// ---------- recipe writes (READY only, bounds-checked) ----------
parToggle := GVL_Cmd.mbParRegs[3];
IF (parToggle <> lastParTog) AND (GVL_Sts.mode = E_MachMode.READY) THEN
    lastParTog := parToggle;
    itemP := WORD_TO_INT(GVL_Cmd.mbParRegs[0]);
    cookP := TO_LREAL(WORD_TO_INT(GVL_Cmd.mbParRegs[1])) / 10.0;
    setP  := TO_LREAL(WORD_TO_INT(GVL_Cmd.mbParRegs[2])) / 10.0;
    IF (itemP >= 1) AND (itemP <= 4)
       AND (cookP >= 20.0) AND (cookP <= 300.0)
       AND (setP >= 120.0) AND (setP <= 230.0) THEN
        GVL_Par.aRecipe[itemP].cookTimeS  := cookP;
        GVL_Par.aRecipe[itemP].platenSetC := setP;
    END_IF
END_IF

END_PROGRAM

// Device/Application/05_L4_Comms/PRG_HMI
(* ============================================================
   PRG_HMI — HMI request edges + password-gated jog (T_Comms).
   Buttons arrive as GVL_Cmd.hmi* (mapped to HMI tags at site).
   NOTE: in the SFC/LD refactor this POU's edge networks become
   LD rungs one-per-button (technician-facing).
   ============================================================ *)
PROGRAM PRG_HMI
VAR
    rtStart, rtStop, rtReset, rtAck, rtClean : R_TRIG;
    jogPermit : BOOL;
    jogStep   : LREAL;
    tonJog    : TON;
    MAINT_PIN : UINT := 2468;   // TODO site-specific, move to secure store
    rtRecW, rtTrimW : R_TRIG;
    recOk   : BOOL;
    recIt   : INT;
    recV    : LREAL;
    trimP   : INT;
    bJogP, bJogM : BOOL;         // jog levels (direct var OR HMI register bit)
    wFlags  : WORD;
    it2, z2, base : INT;
    rtPrsW  : R_TRIG;            // press service command
    prsSel  : INT;
    prsHold : INT;               // holds CmdExec for a few comms cycles
    prsView : INT;               // press shown on the status page
END_VAR

// ---------- LT2100E register unpack (HMI writes %MW600..609) ----------
// reg[0] button bits: 0=start 1=stop 2=reset 3=ack 4=clean
//                     5=jog+ 6=jog- 7=recipeWrite 8=trimWrite
// Numerics are copied only while their write/jog bit is held, so direct
// variable writes (watch list / sim testing) keep working unchanged.
IF GVL_Cmd.hmiRegsCmd[1] <> 0 THEN
    GVL_Cmd.hmiMaintPin := TO_UINT(GVL_Cmd.hmiRegsCmd[1]);
END_IF
IF (GVL_Cmd.hmiRegsCmd[0] AND 16#0060) <> 0 THEN            // a jog bit is held
    GVL_Cmd.hmiJogAxis := TO_INT(GVL_Cmd.hmiRegsCmd[2]);
END_IF
IF (GVL_Cmd.hmiRegsCmd[0] AND 16#0080) <> 0 THEN            // recipe write
    GVL_Cmd.hmiRecItem  := TO_UINT(GVL_Cmd.hmiRegsCmd[3]);
    GVL_Cmd.hmiRecField := TO_UINT(GVL_Cmd.hmiRegsCmd[4]);
    GVL_Cmd.hmiRecValue := TO_LREAL(GVL_Cmd.hmiRegsCmd[5]) / 10.0;   // x10 scaling
END_IF
IF (GVL_Cmd.hmiRegsCmd[0] AND 16#0100) <> 0 THEN            // trim write
    GVL_Cmd.hmiTrimPress := TO_UINT(GVL_Cmd.hmiRegsCmd[6]);
    GVL_Cmd.hmiTrimDelta := TO_LREAL(TO_INT(GVL_Cmd.hmiRegsCmd[7])) / 100.0;  // x100 signed
END_IF
bJogP := GVL_Cmd.hmiJogPlus  OR ((GVL_Cmd.hmiRegsCmd[0] AND 16#0020) <> 0);
bJogM := GVL_Cmd.hmiJogMinus OR ((GVL_Cmd.hmiRegsCmd[0] AND 16#0040) <> 0);

rtStart(CLK := GVL_Cmd.hmiStart OR ((GVL_Cmd.hmiRegsCmd[0] AND 16#0001) <> 0));
rtStop (CLK := GVL_Cmd.hmiStop  OR ((GVL_Cmd.hmiRegsCmd[0] AND 16#0002) <> 0));
rtReset(CLK := GVL_Cmd.hmiReset OR ((GVL_Cmd.hmiRegsCmd[0] AND 16#0004) <> 0));
rtAck  (CLK := GVL_Cmd.hmiAck   OR ((GVL_Cmd.hmiRegsCmd[0] AND 16#0008) <> 0));
rtClean(CLK := GVL_Cmd.hmiClean OR ((GVL_Cmd.hmiRegsCmd[0] AND 16#0010) <> 0));

GVL_Cmd.reqStart  := rtStart.Q;
GVL_Cmd.reqStop   := rtStop.Q  OR GVL_Cmd.reqStop;    // JobExec may also set; consumed by Supervisor edge
GVL_Cmd.reqReset  := rtReset.Q;
GVL_Cmd.reqAckAll := rtAck.Q;
GVL_Cmd.reqClean  := rtClean.Q OR GVL_Cmd.reqClean;
// self-clearing one-shot semantics: Supervisor uses R_TRIG on these,
// so clear them after one comms cycle
IF NOT rtStop.Q  THEN GVL_Cmd.reqStop  := FALSE; END_IF
IF NOT rtClean.Q THEN GVL_Cmd.reqClean := FALSE; END_IF

// ---------- jog (maintenance only) ----------
jogPermit := (GVL_Cmd.hmiMaintPin = MAINT_PIN)
         AND ((GVL_Sts.mode = E_MachMode.READY) OR (GVL_Sts.mode = E_MachMode.FAULT))
         AND GVL_Sts.safetyOk;
tonJog(IN := jogPermit AND (bJogP OR bJogM), PT := T#100MS);
IF tonJog.Q THEN
    tonJog(IN := FALSE);
    jogStep := LIMIT(1.0, GVL_Par.jogVel, GVL_Cfg.JOG_VEL_MAX) * 0.1;  // mm per 100 ms
    IF bJogM THEN jogStep := -jogStep; END_IF
    CASE GVL_Cmd.hmiJogAxis OF
        1: IF NOT GVL_Mech.axGX.Busy THEN
               GVL_Mech.axGX.TargetPos := GVL_Mech.axGX.Sts.actPos + jogStep;
               GVL_Mech.axGX.Vel := GVL_Par.jogVel;
               GVL_Mech.axGX.MoveExec := TRUE;
           END_IF
        2: IF NOT GVL_Mech.axGT.Busy THEN
               GVL_Mech.axGT.TargetPos := GVL_Mech.axGT.Sts.actPos + jogStep;
               GVL_Mech.axGT.Vel := GVL_Par.jogVel;
               GVL_Mech.axGT.MoveExec := TRUE;
           END_IF
        3: IF NOT GVL_Mech.axGZ.Busy THEN
               GVL_Mech.axGZ.TargetPos := GVL_Mech.axGZ.Sts.actPos + jogStep;
               GVL_Mech.axGZ.Vel := GVL_Par.jogVel;
               GVL_Mech.axGZ.MoveExec := TRUE;
           END_IF
        // axes 4..8: same pattern for scraper X/Y/Z, fork Z/tele — add as needed
    END_CASE
ELSIF NOT (bJogP OR bJogM) THEN
    GVL_Mech.axGX.MoveExec := FALSE;
    GVL_Mech.axGT.MoveExec := FALSE;
    GVL_Mech.axGZ.MoveExec := FALSE;
END_IF

// ---------- press jog (jog axis select 9 = selected press drive) ----------
// Level-driven; the drive FB only jogs while fully idle. Velocity = Pr6.00.
IF (GVL_Cmd.hmiJogAxis = 9) AND jogPermit THEN
    GVL_Mech.drvPress[TO_INT(LIMIT(0, GVL_Cmd.hmiPressSel, 3))].JogPlus  := bJogP;
    GVL_Mech.drvPress[TO_INT(LIMIT(0, GVL_Cmd.hmiPressSel, 3))].JogMinus := bJogM;
ELSE
    FOR it2 := 0 TO 3 DO
        GVL_Mech.drvPress[it2].JogPlus  := FALSE;
        GVL_Mech.drvPress[it2].JogMinus := FALSE;
    END_FOR
END_IF

// ---------- recipe editor (bounds-checked; rejected while RUN) ----------
rtRecW(CLK := GVL_Cmd.hmiRecWrite OR ((GVL_Cmd.hmiRegsCmd[0] AND 16#0080) <> 0));
IF rtRecW.Q THEN
    GVL_Cmd.hmiRecAck := FALSE; GVL_Cmd.hmiRecErr := FALSE;
    recIt := TO_INT(GVL_Cmd.hmiRecItem);
    recV  := GVL_Cmd.hmiRecValue;
    recOk := (recIt >= 1) AND (recIt <= 4) AND (GVL_Sts.mode <> E_MachMode.RUN);
    IF recOk THEN
        CASE GVL_Cmd.hmiRecField OF
            1: IF (recV >= GVL_Cfg.REC_COOK_MIN)  AND (recV <= GVL_Cfg.REC_COOK_MAX)
               THEN GVL_Par.aRecipe[recIt].cookTimeS := recV;  ELSE recOk := FALSE; END_IF
            2: IF (recV >= GVL_Cfg.REC_SMDUR_MIN) AND (recV <= GVL_Cfg.REC_SMDUR_MAX)
               THEN GVL_Par.aRecipe[recIt].smashDurS := recV;  ELSE recOk := FALSE; END_IF
            3: IF (recV >= GVL_Cfg.REC_SMPOS_MIN) AND (recV <= GVL_Cfg.REC_SMPOS_MAX)
               THEN GVL_Par.aRecipe[recIt].smashPosMm := recV; ELSE recOk := FALSE; END_IF
            4: IF (recV >= GVL_Cfg.REC_HLPOS_MIN) AND (recV <= GVL_Cfg.REC_HLPOS_MAX)
               THEN GVL_Par.aRecipe[recIt].holdPosMm := recV;  ELSE recOk := FALSE; END_IF
            5: IF (recV >= GVL_Cfg.REC_PLSET_MIN) AND (recV <= GVL_Cfg.REC_PLSET_MAX)
               THEN GVL_Par.aRecipe[recIt].platenSetC := recV; ELSE recOk := FALSE; END_IF
        ELSE
            recOk := FALSE;
        END_CASE
        // physical sanity: hold gap must not be tighter than smash gap
        IF recOk AND (GVL_Par.aRecipe[recIt].holdPosMm < GVL_Par.aRecipe[recIt].smashPosMm) THEN
            GVL_Par.aRecipe[recIt].holdPosMm := GVL_Par.aRecipe[recIt].smashPosMm;
        END_IF
    END_IF
    GVL_Cmd.hmiRecAck := recOk;
    GVL_Cmd.hmiRecErr := NOT recOk;
END_IF

// ---------- press calibration trim (maintenance PIN; not while RUN) ----------
rtTrimW(CLK := GVL_Cmd.hmiTrimWrite OR ((GVL_Cmd.hmiRegsCmd[0] AND 16#0100) <> 0));
IF rtTrimW.Q THEN
    GVL_Cmd.hmiTrimAck := FALSE; GVL_Cmd.hmiTrimErr := FALSE;
    trimP := TO_INT(GVL_Cmd.hmiTrimPress);
    IF (trimP >= 0) AND (trimP <= 3)
       AND (GVL_Cmd.hmiMaintPin = MAINT_PIN)
       AND (GVL_Sts.mode <> E_MachMode.RUN)
       AND (ABS(GVL_Cmd.hmiTrimDelta) <= GVL_Cfg.PRESS_TRIM_MAX_MM) THEN
        GVL_Par.pressTrimMm[trimP] := LIMIT(-GVL_Cfg.PRESS_TRIM_MAX_MM,
            GVL_Par.pressTrimMm[trimP] + GVL_Cmd.hmiTrimDelta,
            GVL_Cfg.PRESS_TRIM_MAX_MM);
        GVL_Cmd.hmiTrimAck := TRUE;
    ELSE
        GVL_Cmd.hmiTrimErr := TRUE;
    END_IF
END_IF

// ---------- press service commands (PIN; READY only; press must be idle) ----------
// HMI: reg608 = command (1 HOME, 2 OPEN, 3 PROFILE), reg609 = press 0..3,
// button bit 9 executes. Do not use while the test suite or Gateway runs.
rtPrsW(CLK := GVL_Cmd.hmiPressWrite OR ((GVL_Cmd.hmiRegsCmd[0] AND 16#0200) <> 0));
IF rtPrsW.Q THEN
    GVL_Cmd.hmiPressAck := FALSE; GVL_Cmd.hmiPressErr := FALSE;
    IF (GVL_Cmd.hmiRegsCmd[0] AND 16#0200) <> 0 THEN
        GVL_Cmd.hmiPressCmd := TO_UINT(GVL_Cmd.hmiRegsCmd[8]);
        GVL_Cmd.hmiPressSel := TO_UINT(GVL_Cmd.hmiRegsCmd[9]);
    END_IF
    prsSel := TO_INT(GVL_Cmd.hmiPressSel);
    IF (prsSel >= 0) AND (prsSel <= 3)
       AND (GVL_Cmd.hmiMaintPin = MAINT_PIN)
       AND (GVL_Sts.mode = E_MachMode.READY)
       AND (NOT GVL_Mech.fbPress[prsSel].Busy)
       AND (NOT GVL_Cmd.testStart) THEN
        CASE GVL_Cmd.hmiPressCmd OF
            1: GVL_Mech.fbPress[prsSel].Cmd.code := GVL_Cfg.MCMD_HOME;
               GVL_Cmd.hmiPressAck := TRUE;
            2: GVL_Mech.fbPress[prsSel].Cmd.code := GVL_Cfg.MCMD_OPEN;
               GVL_Cmd.hmiPressAck := TRUE;
            3: IF GVL_Mech.fbPress[prsSel].IsOpen THEN   // profile only from open
                   GVL_Mech.fbPress[prsSel].Recipe :=
                       GVL_Par.aRecipe[LIMIT(1, TO_INT(GVL_Cmd.hmiRecItem), 4)];
                   GVL_Mech.fbPress[prsSel].Cmd.code := GVL_Cfg.MCMD_PROFILE;
                   GVL_Cmd.hmiPressAck := TRUE;
               ELSE
                   GVL_Cmd.hmiPressErr := TRUE;          // open (cmd 2) first
               END_IF
        ELSE
            GVL_Cmd.hmiPressErr := TRUE;
        END_CASE
        IF GVL_Cmd.hmiPressAck THEN
            GVL_Mech.fbPress[prsSel].CmdExec := TRUE;
            prsHold := 3;                    // release after ~3 comms cycles
        END_IF
    ELSE
        GVL_Cmd.hmiPressErr := TRUE;
    END_IF
END_IF
IF prsHold > 0 THEN
    prsHold := prsHold - 1;
    IF prsHold = 0 THEN
        GVL_Mech.fbPress[TO_INT(LIMIT(0, GVL_Cmd.hmiPressSel, 3))].CmdExec := FALSE;
    END_IF
END_IF

// ---------- LT2100E status pack (HMI reads %MW620..669) ----------
GVL_Cmd.hmiRegsSts[0] := TO_WORD(TO_UINT(GVL_Sts.mode));
wFlags := 0;
IF GVL_Cmd.hmiRecAck    THEN wFlags := wFlags OR 16#0001; END_IF
IF GVL_Cmd.hmiRecErr    THEN wFlags := wFlags OR 16#0002; END_IF
IF GVL_Cmd.hmiTrimAck   THEN wFlags := wFlags OR 16#0004; END_IF
IF GVL_Cmd.hmiTrimErr   THEN wFlags := wFlags OR 16#0008; END_IF
IF GVL_Sts.heatAtSet    THEN wFlags := wFlags OR 16#0010; END_IF
IF GVL_Sts.fridgeAtSet  THEN wFlags := wFlags OR 16#0020; END_IF
IF GVL_Sts.allHomed     THEN wFlags := wFlags OR 16#0040; END_IF
IF GVL_Sts.safetyOk     THEN wFlags := wFlags OR 16#0080; END_IF
IF GVL_Sts.cleanCoolOk  THEN wFlags := wFlags OR 16#0100; END_IF
IF GVL_Cmd.hmiPressAck  THEN wFlags := wFlags OR 16#0200; END_IF
IF GVL_Cmd.hmiPressErr  THEN wFlags := wFlags OR 16#0400; END_IF
GVL_Cmd.hmiRegsSts[1] := wFlags;
GVL_Cmd.hmiRegsSts[2] := TO_WORD(TO_UINT(GVL_Alm.nActive));
GVL_Cmd.hmiRegsSts[3] := TO_WORD(GVL_Alm.aActive[0].id AND 16#FFFF);          // code
GVL_Cmd.hmiRegsSts[4] := TO_WORD(SHR(GVL_Alm.aActive[0].id, 16) AND 16#FFFF); // subsystem
GVL_Cmd.hmiRegsSts[5] := TO_WORD(TO_UINT(GVL_Sts.uptimeS MOD 65536));
// griddle states 626..629
FOR z2 := 0 TO 3 DO
    GVL_Cmd.hmiRegsSts[6 + z2] := TO_WORD(GVL_Sts.aGriddle[z2].state);
END_FOR
// recipe readback 630..649: per item 1..4 -> cook, smashDur, smashPos, holdPos, platenSet (all x10)
FOR it2 := 1 TO 4 DO
    base := 10 + (it2 - 1) * 5;
    GVL_Cmd.hmiRegsSts[base]     := TO_WORD(TO_UINT(GVL_Par.aRecipe[it2].cookTimeS  * 10.0));
    GVL_Cmd.hmiRegsSts[base + 1] := TO_WORD(TO_UINT(GVL_Par.aRecipe[it2].smashDurS  * 10.0));
    GVL_Cmd.hmiRegsSts[base + 2] := TO_WORD(TO_UINT(GVL_Par.aRecipe[it2].smashPosMm * 10.0));
    GVL_Cmd.hmiRegsSts[base + 3] := TO_WORD(TO_UINT(GVL_Par.aRecipe[it2].holdPosMm  * 10.0));
    GVL_Cmd.hmiRegsSts[base + 4] := TO_WORD(TO_UINT(GVL_Par.aRecipe[it2].platenSetC * 10.0));
END_FOR
// press trims 650..653 (x100 signed)
FOR z2 := 0 TO 3 DO
    GVL_Cmd.hmiRegsSts[30 + z2] := TO_WORD(TO_INT(GVL_Par.pressTrimMm[z2] * 100.0));
END_FOR
// temperatures 654..661 platens, 662 fridge (x10)
FOR z2 := 0 TO 7 DO
    GVL_Cmd.hmiRegsSts[34 + z2] := TO_WORD(TO_INT(GVL_Sts.aHeat[z2].actC * 10.0));
END_FOR
GVL_Cmd.hmiRegsSts[42] := TO_WORD(TO_INT(GVL_Sts.fridgeActC * 10.0));
// press service status page 663..667 (selected press)
prsView := TO_INT(LIMIT(0, GVL_Cmd.hmiPressSel, 3));
GVL_Cmd.hmiRegsSts[43] := TO_WORD(GVL_Mech.fbPress[prsView].State);
wFlags := 0;
IF GVL_Mech.drvPress[prsView].Homed    THEN wFlags := wFlags OR 16#0001; END_IF
IF GVL_Mech.fbPress[prsView].IsOpen    THEN wFlags := wFlags OR 16#0002; END_IF
IF GVL_Mech.fbPress[prsView].Holding   THEN wFlags := wFlags OR 16#0004; END_IF
IF GVL_Mech.fbPress[prsView].Busy      THEN wFlags := wFlags OR 16#0008; END_IF
IF GVL_Mech.fbPress[prsView].Error     THEN wFlags := wFlags OR 16#0010; END_IF
IF GVL_Mech.drvPress[prsView].HomeBusy THEN wFlags := wFlags OR 16#0020; END_IF
IF GVL_Mech.drvPress[prsView].ParamsValid THEN wFlags := wFlags OR 16#0040; END_IF
IF GVL_Mech.drvPress[prsView].Busy     THEN wFlags := wFlags OR 16#0080; END_IF
GVL_Cmd.hmiRegsSts[44] := wFlags;
GVL_Cmd.hmiRegsSts[45] := GVL_IO.iMbPrStatus;   // bench drive raw status word
GVL_Cmd.hmiRegsSts[46] := TO_WORD(GVL_Mech.fbPress[prsView].ErrorID AND 16#FFFF);
GVL_Cmd.hmiRegsSts[47] := TO_WORD(SHR(GVL_Mech.fbPress[prsView].ErrorID, 16) AND 16#FFFF);
// jog feedback 668: selected axis actual position, mm/deg x10 (signed)
CASE GVL_Cmd.hmiJogAxis OF
    1: GVL_Cmd.hmiRegsSts[48] := TO_WORD(TO_INT(GVL_Mech.axGX.Sts.actPos * 10.0));
    2: GVL_Cmd.hmiRegsSts[48] := TO_WORD(TO_INT(GVL_Mech.axGT.Sts.actPos * 10.0));
    3: GVL_Cmd.hmiRegsSts[48] := TO_WORD(TO_INT(GVL_Mech.axGZ.Sts.actPos * 10.0));
ELSE
    GVL_Cmd.hmiRegsSts[48] := 0;
END_CASE

END_PROGRAM

// Device/Application/02_L1_Drivers/FB_AxisCtrl
(* ============================================================
   FB_AxisCtrl — single-axis wrapper. The ONLY POU calling MC_*.
   Runs in T_Motion. One instance per axis, body called EVERY cycle.
   SIM: internal kinematic model (trapezoid-less: const-vel ramp).
   REAL: SoftMotion CiA-402 via SM3_Basic.
   ============================================================ *)
FUNCTION_BLOCK FB_AxisCtrl
VAR_INPUT
    Sim       : BOOL;
    SubsysId  : UINT;
    Enable    : BOOL;
    HomeExec  : BOOL;          // level; internally edge-latched
    MoveExec  : BOOL;
    TargetPos : LREAL;
    Vel       : LREAL := 100.0;
    Acc       : LREAL := 500.0;
    StopExec  : BOOL;
    ResetExec : BOOL;
    Abort     : BOOL;
    CycleMs   : LREAL := 4.0;
    SimHomeS  : LREAL := 1.0;  // sim homing duration
END_VAR
VAR_IN_OUT
    Axis : AXIS_REF_SM3;
END_VAR
VAR_OUTPUT
    Sts     : ST_AxisSts;
    Busy    : BOOL;
    Done    : BOOL;            // latched until next exec
    Error   : BOOL;
    ErrorID : UDINT;
END_VAR
VAR
    state     : INT;           // 0 idle 1 homing 2 moving 3 stopping
    rtHome, rtMove, rtReset : R_TRIG;
    tonTO     : TON;
    // sim model
    simPos    : LREAL;
    simTgt    : LREAL;
    simHomeT  : LREAL;
    // real motion FBs
    mcPower   : MC_Power;
    mcHome    : MC_Home;
    mcMove    : MC_MoveAbsolute;
    mcStop    : MC_Stop;
    mcReset   : MC_Reset;
    dtS       : LREAL;
    stepMax   : LREAL;
END_VAR


dtS := CycleMs / 1000.0;
rtHome(CLK := HomeExec);
rtMove(CLK := MoveExec);
rtReset(CLK := ResetExec);

IF Abort THEN
    state := 0; Busy := FALSE;
    tonTO(IN := FALSE);
END_IF

IF rtReset.Q THEN
    Error := FALSE; ErrorID := 0;
END_IF

IF Sim THEN
    // ---------------- SIMULATION MODEL ----------------
    Sts.powered := Enable;
    CASE state OF
        0: // idle
            IF Enable AND rtHome.Q THEN
                state := 1; simHomeT := 0.0; Busy := TRUE; Done := FALSE;
            ELSIF Enable AND Sts.homed AND rtMove.Q THEN
                simTgt := TargetPos; state := 2; Busy := TRUE; Done := FALSE;
                tonTO(IN := FALSE);
            ELSIF Enable AND (NOT Sts.homed) AND rtMove.Q THEN
                Error := TRUE; ErrorID := F_Err(SubsysId, GVL_Cfg.ERR_NOT_HOMED);
            END_IF
        1: // homing
            simHomeT := simHomeT + dtS;
            IF simHomeT >= SimHomeS THEN
                simPos := 0.0; Sts.homed := TRUE;
                state := 0; Busy := FALSE; Done := TRUE;
            END_IF
        2: // moving: constant-velocity approach
            stepMax := Vel * dtS;
            IF ABS(simTgt - simPos) <= stepMax THEN
                simPos := simTgt;
                state := 0; Busy := FALSE; Done := TRUE;
            ELSIF simTgt > simPos THEN
                simPos := simPos + stepMax;
            ELSE
                simPos := simPos - stepMax;
            END_IF
            tonTO(IN := TRUE, PT := GVL_Cfg.TO_AXIS_MOVE);
            IF tonTO.Q THEN
                state := 0; Busy := FALSE; Error := TRUE;
                ErrorID := F_Err(SubsysId, GVL_Cfg.ERR_TIMEOUT);
            END_IF
    END_CASE
    IF StopExec THEN state := 0; Busy := FALSE; END_IF
    Sts.actPos := simPos;
    Sts.inPos  := (state = 0);
ELSE
    // ---------------- REAL HARDWARE (SoftMotion) ----------------
    mcPower(Axis := Axis, Enable := Enable, bRegulatorOn := Enable, bDriveStart := Enable);
    Sts.powered := mcPower.Status;

    mcHome(Axis := Axis, Execute := (rtHome.Q OR mcHome.Busy) AND NOT Abort, Position := 0.0);
    IF mcHome.Done THEN Sts.homed := TRUE; END_IF

    mcMove(Axis := Axis,
           Execute      := (rtMove.Q OR mcMove.Busy) AND NOT Abort AND NOT StopExec,
           Position     := TargetPos,
           Velocity     := Vel,
           Acceleration := Acc,
           Deceleration := Acc);

    mcStop(Axis := Axis, Execute := StopExec OR Abort, Deceleration := Acc * 2.0);
    mcReset(Axis := Axis, Execute := rtReset.Q);

    Busy := mcHome.Busy OR mcMove.Busy;
    IF mcHome.Done OR mcMove.Done THEN Done := TRUE; END_IF
    IF rtHome.Q OR rtMove.Q THEN Done := FALSE; END_IF

    IF mcMove.Error OR mcHome.Error OR mcPower.Error THEN
        Error := TRUE;
        ErrorID := F_Err(SubsysId, GVL_Cfg.ERR_DRIVE);
        Sts.homed := FALSE;              // demand re-home after drive fault
    END_IF
    Sts.actPos := Axis.fSetPosition;     // TODO: use MC_ReadActualPosition if preferred
    Sts.inPos  := NOT Busy;
END_IF

IF NOT Sts.powered THEN Sts.homed := FALSE; END_IF   // power loss clears homed
Sts.errorId := ErrorID;

END_FUNCTION_BLOCK

// Device/Application/02_L1_Drivers/FB_PidHeater
(* ============================================================
   FB_PidHeater — PI + time-proportioned SSR + TC plausibility.
   Call every T_App cycle; internal divider executes PI at 100 ms.
   SIM: first-order plant  dT = (gain*out - (T-Tamb)/tau) * dt
   Independent hardwired thermostat is the REAL protection; the
   over-temp check here is early warning (INFO/ZONE only).
   ============================================================ *)
FUNCTION_BLOCK FB_PidHeater
VAR_INPUT
    Sim          : BOOL;
    ZoneId       : INT;          // 0..7
    Enable       : BOOL;
    SetC         : LREAL := 200.0;
    iTempRaw     : INT;          // 0.1 degC from TC module
    StaggerToken : BOOL;         // may ramp (from FB_HeatBank)
    CycleMs      : LREAL := 20.0;
END_VAR
VAR_OUTPUT
    qSsr    : BOOL;
    Zone    : ST_HeatZone;
    Error   : BOOL;
    ErrorID : UDINT;
END_VAR
VAR
    divCnt   : INT;
    actC     : LREAL;
    lastC    : LREAL;
    err      : LREAL;
    integ    : LREAL;
    outPct   : LREAL;
    pwmT     : LREAL;
    simC     : LREAL := 25.0;
    dtPi     : LREAL := 0.1;
    tcFaultCnt : INT;
    SIM_GAIN : LREAL := 3.5;     // degC/s at 100 %
    SIM_TAU  : LREAL := 60.0;
    ramping  : BOOL;
END_VAR

// ---- acquire temperature ----
IF Sim THEN
    simC := simC + (SIM_GAIN * outPct / 100.0 - (simC - 25.0) / SIM_TAU)
                 * (CycleMs / 1000.0) * GVL_Cfg.SIM_TIME_SCALE;
    actC := simC;
ELSE
    actC := TO_LREAL(iTempRaw) / 10.0;
END_IF

// ---- TC plausibility (real only) ----
IF NOT Sim THEN
    IF (actC < -20.0) OR (actC > 400.0) THEN tcFaultCnt := tcFaultCnt + 1; ELSE tcFaultCnt := 0; END_IF
    IF ABS(actC - lastC) > GVL_Cfg.TC_RATE_MAX * (CycleMs / 1000.0) * 10.0 THEN
        tcFaultCnt := tcFaultCnt + 1;
    END_IF
    IF tcFaultCnt > 25 THEN
        Error := TRUE;
        ErrorID := F_Err(GVL_Cfg.SS_HEAT_0 + TO_UINT(ZoneId), GVL_Cfg.ERR_TC);
    END_IF
END_IF
lastC := actC;

// ---- PI @100 ms ----
divCnt := divCnt + 1;
IF divCnt >= 5 THEN
    divCnt := 0;
    ramping := (SetC - actC) > 20.0;
    IF Enable AND NOT Error AND (StaggerToken OR NOT ramping) THEN
        err := SetC - actC;
        integ := LIMIT(0.0, integ + err * GVL_Cfg.HEAT_KI * dtPi * 100.0, 100.0);
        outPct := LIMIT(0.0, GVL_Cfg.HEAT_KP * err + integ, 100.0);
    ELSE
        outPct := 0.0; integ := 0.0;
    END_IF
END_IF

// ---- time-proportioned SSR ----
pwmT := pwmT + CycleMs;
IF pwmT >= GVL_Cfg.PWM_WINDOW_MS THEN pwmT := 0.0; END_IF
qSsr := Enable AND NOT Error AND (pwmT < outPct / 100.0 * GVL_Cfg.PWM_WINDOW_MS);

Zone.setC := SetC;   Zone.actC := actC;   Zone.outPct := outPct;
Zone.tcOk := NOT Error;
Zone.atSet := ABS(SetC - actC) <= GVL_Cfg.HEAT_AT_BAND;
Zone.enabled := Enable;

END_FUNCTION_BLOCK

// Device/Application/03_L2_Mechanisms/FB_HeatBank
(* ============================================================
   FB_HeatBank — supervises 8 FB_PidHeater zones: stagger tokens
   (inrush cap during ramp) + aggregate status. Call AFTER the
   heater bodies each T_App cycle (one-cycle token lag is fine).
   Zone map: griddle g -> zones 2g (top), 2g+1 (bottom).
   ============================================================ *)
FUNCTION_BLOCK FB_HeatBank
VAR_INPUT
    Enable : BOOL;
END_VAR
VAR_IN_OUT
    Heaters : ARRAY[0..7] OF FB_PidHeater;
END_VAR
VAR_OUTPUT
    Token    : ARRAY[0..7] OF BOOL;
    AllAtSet : BOOL;
    MaxDevC  : LREAL;
    AnyTcErr : BOOL;
END_VAR
VAR
    z        : INT;
    nRamping : INT;
    ramping  : BOOL;
    dev      : LREAL;
END_VAR

nRamping := 0; AllAtSet := Enable; MaxDevC := 0.0; AnyTcErr := FALSE;
FOR z := 0 TO 7 DO
    ramping := (Heaters[z].Zone.setC - Heaters[z].Zone.actC) > 20.0;
    IF ramping THEN
        IF nRamping < GVL_Cfg.HEAT_MAX_STAGGER THEN
            Token[z] := TRUE; nRamping := nRamping + 1;
        ELSE
            Token[z] := FALSE;
        END_IF
    ELSE
        Token[z] := TRUE;   // regulation always allowed
    END_IF
    dev := ABS(Heaters[z].Zone.setC - Heaters[z].Zone.actC);
    IF dev > MaxDevC THEN MaxDevC := dev; END_IF
    IF NOT Heaters[z].Zone.atSet THEN AllAtSet := FALSE; END_IF
    IF Heaters[z].Error THEN AnyTcErr := TRUE; END_IF
END_FOR
IF NOT Enable THEN AllAtSet := FALSE; END_IF

END_FUNCTION_BLOCK

// Device/Application/02_L1_Drivers/FB_PneuActuator
(* ============================================================
   FB_PneuActuator — valve + 2 reed/prox sensors + timeout.
   Cmd TRUE = extend/open, FALSE = retract/close.
   Runs in T_App. SIM: sensors flip after SIM_TRAVEL_S.
   ============================================================ *)
FUNCTION_BLOCK FB_PneuActuator
VAR_INPUT
    Sim        : BOOL;
    SubsysId   : UINT;
    Cmd        : BOOL;
    iExtended  : BOOL;
    iRetracted : BOOL;
    CycleMs    : LREAL := 20.0;
END_VAR
VAR_OUTPUT
    qValve    : BOOL;
    Extended  : BOOL;
    Retracted : BOOL;
    Moving    : BOOL;
    Error     : BOOL;
    ErrorID   : UDINT;
END_VAR
VAR
    tonTO   : TON;
    lastCmd : BOOL;
    simT    : LREAL;
    simExt  : BOOL;
    SIM_TRAVEL_S : LREAL := 0.3;
    extEff, retEff : BOOL;
END_VAR


qValve := Cmd;
IF Cmd <> lastCmd THEN
    simT := 0.0;
    lastCmd := Cmd;
END_IF

IF Sim THEN
    simT := simT + CycleMs / 1000.0;
    IF simT >= SIM_TRAVEL_S THEN simExt := Cmd; END_IF
    extEff := simExt;  retEff := NOT simExt;
ELSE
    extEff := iExtended; retEff := iRetracted;
END_IF

IF extEff AND retEff THEN                 // both sensors -> wiring fault
    Error := TRUE; ErrorID := F_Err(SubsysId, GVL_Cfg.ERR_SENSOR);
END_IF

Extended  := extEff AND NOT retEff;
Retracted := retEff AND NOT extEff;
Moving    := NOT Extended AND NOT Retracted;

tonTO(IN := (Cmd AND NOT Extended) OR (NOT Cmd AND NOT Retracted), PT := GVL_Cfg.TO_PNEU);
IF tonTO.Q THEN
    Error := TRUE; ErrorID := F_Err(SubsysId, GVL_Cfg.ERR_TIMEOUT);
END_IF

END_FUNCTION_BLOCK

// Device/Application/02_L1_Drivers/FB_PressDrive
(* ============================================================
   FB_PressDrive — CS2RS in PR mode, DI-trigger control.
   Validated pattern from the gantry test project:
     - set path-select DOs, wait one cycle, raise CTRG and HOLD it
       until InPos confirms (never a single-scan pulse)
     - InPos handshake = "saw moving" (InPos drops, then returns)
   Modbus RTU monitoring (position/alarm) is DIAGNOSTIC ONLY and
   added at migration (stub hooks below). Runs in T_App (20 ms).
   PR paths (configure in drive, MIGRATION_GUIDE step 4):
     path 0 = OPEN position, path 1 = SMASH pos, path 2 = HOLD pos
   ============================================================ *)
FUNCTION_BLOCK FB_PressDrive
VAR_INPUT
    Sim      : BOOL;
    SubsysId : UINT;
    Enable   : BOOL;
    PathExec : BOOL;             // edge latches PathNo
    PathNo   : INT;              // 0..2
    Abort    : BOOL;
    iInPos   : BOOL;             // from drive DO (via IoMap)
    iAlarm   : BOOL;
    CycleMs  : LREAL := 20.0;
    // PR path table parameterization (positions written to drive before use)
    OpenPosMm  : LREAL := 60.0;  // path 0
    SmashPosMm : LREAL := 4.0;   // path 1
    HoldPosMm  : LREAL := 6.0;   // path 2
    WriteParams : BOOL;          // edge: push the 3 positions to the drive
    // Modbus transport feedback (wired from the NetworkConfig channel glue)
    MbWrDone : BOOL;             // transport confirms last write
    MbWrErr  : BOOL;             // transport reports failure
    // homing (real: Modbus 0x0020 -> 0x6002; done = status bit 0x40)
    HomeExec    : BOOL;          // edge: re-reference the drive
    MbHomeDone  : BOOL;          // home-channel transport ack
    iStatusWord : WORD;          // cyclic 0x1003 image (glue; 0 in sim)
    // maintenance jog (real: 0x4001/0x4002 -> 0x1801; velocity = drive Pr6.00)
    JogPlus, JogMinus : BOOL;    // level; only acts while drive fully idle
    MbJogDone : BOOL;            // jog-channel transport ack
END_VAR
VAR_OUTPUT
    qSel0, qSel1, qCtrg, qEnable : BOOL;
    Busy, Done, Error : BOOL;
    ErrorID : UDINT;
    ActPath : INT := -1;
    // parameter channel status
    ParamsValid : BOOL;          // drive path table matches last written values
    ParamBusy   : BOOL;
    ParamErr    : BOOL;
    // Modbus write request (routed to a NetworkConfig write channel by glue)
    MbPath   : INT;              // which PR path's position is being written (0..2)
    MbValH   : WORD;             // position high word
    MbValL   : WORD;             // position low word
    MbWrExec : BOOL;             // held TRUE until MbWrDone/MbWrErr
    // homing status/request
    Homed      : BOOL;           // drive is referenced (sim: always TRUE)
    HomeBusy   : BOOL;           // homing sequence in progress
    MbHomeExec : BOOL;           // trigger for the home write channel
    // jog request (routed to the jog write channel)
    MbJogVal   : WORD;           // 16#4001 = jog+, 16#4002 = jog-
    MbJogExec  : BOOL;
END_VAR
VAR
    state    : INT;
    rtExec   : R_TRIG;
    latched  : INT;
    sawMoving: BOOL;
    tonTO    : TON;
    inPosEff : BOOL;
    // sim
    simTimer : LREAL;
    SIM_TRAVEL_S : LREAL := 0.8;
    // param write channel
    rtWr     : R_TRIG;
    pStep    : INT;
    pRetry   : INT;
    P_MAX_RETRY : INT := 3;
    shadowOpen, shadowSmash, shadowHold : LREAL;  // last values confirmed in drive
    pInit    : BOOL;             // at least one successful full push done
    pIdx     : INT;              // 0..2: one write per PR path (posH+posL together)
    pPosMm   : LREAL;
    pPulses  : DINT;
    tonMb    : TON;              // per-transaction timeout
    // homing machine
    rtHome  : R_TRIG;
    hStep   : INT;
    hSaw    : BOOL;              // saw not-homed during the sequence (stale-bit guard)
    tonHome : TON;
    // jog machine
    jStep   : INT;
    tonJog  : TON;
END_VAR


rtExec(CLK := PathExec);
qEnable := Enable;

// effective InPos: sim model or hardware input
IF Sim THEN
    inPosEff := (state <> 3) OR (simTimer >= SIM_TRAVEL_S);
ELSE
    inPosEff := iInPos;
END_IF

IF Abort THEN
    state := 0; Busy := FALSE; qCtrg := FALSE;
    tonTO(IN := FALSE);
END_IF

IF (NOT Sim) AND iAlarm THEN
    Error := TRUE; ErrorID := F_Err(SubsysId, GVL_Cfg.ERR_DRIVE);
    state := 0; Busy := FALSE; qCtrg := FALSE;
    pInit := FALSE;   // drive may have power-cycled: RAM PR table reverts to
                      // EEPROM, so force a full re-push on the next profile
END_IF

CASE state OF
    0: // idle
        qCtrg := FALSE;
        IF Enable AND rtExec.Q AND (PathNo >= 0) AND (PathNo <= 2) THEN
            latched := PathNo;
            qSel0 := (latched MOD 2) = 1;
            qSel1 := ((latched / 2) MOD 2) = 1;
            state := 1; Busy := TRUE; Done := FALSE;
            Error := FALSE; ErrorID := 0;      // new attempt clears a latched error
            sawMoving := FALSE; simTimer := 0.0;
            tonTO(IN := FALSE);
        END_IF
    1: // one full cycle DO settle before CTRG (drive DI filter)
        state := 3;
        qCtrg := TRUE;                     // held high for whole move
    3: // executing: wait saw-moving handshake
        simTimer := simTimer + CycleMs / 1000.0;
        IF NOT inPosEff THEN sawMoving := TRUE; END_IF
        tonTO(IN := TRUE, PT := GVL_Cfg.TO_PRESS);
        // completion: normal = saw-moving handshake; zero-distance = INP never
        // dropped because target == current position (old Z-rig special case)
        IF inPosEff AND (sawMoving OR (Sim AND simTimer >= SIM_TRAVEL_S)
                         OR ((NOT sawMoving) AND (simTimer >= 0.5))) THEN
            qCtrg := FALSE; ActPath := latched;
            state := 0; Busy := FALSE; Done := TRUE;
            tonTO(IN := FALSE);
        ELSIF tonTO.Q THEN
            qCtrg := FALSE;
            state := 0; Busy := FALSE; Error := TRUE;
            ErrorID := F_Err(SubsysId, GVL_Cfg.ERR_TIMEOUT);
        END_IF
END_CASE

// ============================================================
// PR path table parameter writer (positions only; motion stays DI).
// SIM: accepted instantly. HARDWARE: closed-loop Modbus RTU write ->
// readback verify -> retry (pattern proven on the old Z-axis rig).
// Only call while press idle; FB_Press guarantees this.
// ============================================================
rtWr(CLK := WriteParams);
IF rtWr.Q AND (pStep = 0) THEN
    ParamsValid := FALSE; ParamErr := FALSE; ParamBusy := TRUE;
    Error := FALSE; ErrorID := 0;              // new attempt clears a latched error
    pRetry := 0; pStep := 1;
END_IF

CASE pStep OF
    0: ;
    1: // route: skip if drive already holds these values
        IF pInit AND (OpenPosMm = shadowOpen) AND (SmashPosMm = shadowSmash)
                 AND (HoldPosMm = shadowHold) THEN
            ParamsValid := TRUE; ParamBusy := FALSE; pStep := 0;
        ELSIF Sim THEN
            // simulation: accept instantly
            shadowOpen := OpenPosMm; shadowSmash := SmashPosMm; shadowHold := HoldPosMm;
            pInit := TRUE;
            ParamsValid := TRUE; ParamBusy := FALSE; pStep := 0;
        ELSE
            pIdx := 0; pStep := 2;                        // real Modbus push, path by path
        END_IF
    2: // compose path write pIdx (posH+posL in one write-multiple transaction)
        CASE pIdx OF
            0: pPosMm := OpenPosMm;
            1: pPosMm := SmashPosMm;
            2: pPosMm := HoldPosMm;
        END_CASE
        pPulses := TO_DINT(pPosMm * GVL_Cfg.PRESS_PULSES_PER_MM);
        MbPath := pIdx;
        MbValH := TO_WORD(SHR(TO_DWORD(pPulses), 16) AND 16#FFFF);
        MbValL := TO_WORD(TO_DWORD(pPulses) AND 16#FFFF);
        MbWrExec := TRUE; tonMb(IN := FALSE);
        pStep := 3;
    3: // wait channel ack (glue reflects the NetworkConfig channel done/error)
        tonMb(IN := TRUE, PT := T#1S);
        IF MbWrDone THEN
            MbWrExec := FALSE; tonMb(IN := FALSE); pRetry := 0;
            pIdx := pIdx + 1;
            IF pIdx > 2 THEN
                shadowOpen := OpenPosMm; shadowSmash := SmashPosMm; shadowHold := HoldPosMm;
                pInit := TRUE;
                ParamsValid := TRUE; ParamBusy := FALSE; pStep := 0;
            ELSE
                pStep := 2;                               // next path (fresh trigger edge)
            END_IF
        ELSIF MbWrErr OR tonMb.Q THEN
            MbWrExec := FALSE; tonMb(IN := FALSE);
            pRetry := pRetry + 1;
            IF pRetry > P_MAX_RETRY THEN
                ParamErr := TRUE; ParamBusy := FALSE; pStep := 0;
            ELSE
                pStep := 2;                               // resend same path
            END_IF
        END_IF
END_CASE

// ============================================================
// Homing (drive re-reference). Real: write 0x0020 to 0x6002 via the home
// channel, completion = status-word bit 0x40 (with stale-bit guard).
// Sim: always homed. Proven pattern from the old Z-axis rig.
// ============================================================
IF Sim THEN
    Homed := TRUE;
ELSE
    Homed := (iStatusWord AND 16#0040) <> 0;
END_IF
rtHome(CLK := HomeExec);
CASE hStep OF
    0:
        IF rtHome.Q AND NOT Sim THEN
            Error := FALSE; ErrorID := 0;      // new attempt clears a latched error
            MbHomeExec := TRUE; tonHome(IN := FALSE); hStep := 1;
        END_IF
    1: // wait home-channel transport ack
        tonHome(IN := TRUE, PT := T#1S);
        IF MbHomeDone THEN
            MbHomeExec := FALSE; tonHome(IN := FALSE);
            hSaw := FALSE; hStep := 2;
        ELSIF tonHome.Q THEN
            MbHomeExec := FALSE; tonHome(IN := FALSE);
            Error := TRUE; ErrorID := F_Err(SubsysId, GVL_Cfg.ERR_DRIVE);
            hStep := 0;
        END_IF
    2: // wait homing complete (bit drops while homing, then returns)
        tonHome(IN := TRUE, PT := T#30S);
        IF NOT Homed THEN hSaw := TRUE; END_IF
        IF Homed AND (hSaw OR (tonHome.ET >= T#2S)) THEN
            tonHome(IN := FALSE); hStep := 0;
        ELSIF tonHome.Q THEN
            tonHome(IN := FALSE);
            Error := TRUE; ErrorID := F_Err(SubsysId, GVL_Cfg.ERR_TIMEOUT);
            hStep := 0;
        END_IF
END_CASE
HomeBusy := hStep <> 0;

// ============================================================
// Maintenance jog: repeated point-jog writes (0x4001/0x4002 -> 0x1801)
// while the button is held. Real mode only, and ONLY while the drive is
// fully idle (no path, no params, no homing). Velocity = drive Pr6.00.
// ============================================================
IF Sim OR (state <> 0) OR (pStep <> 0) OR (hStep <> 0) OR Busy THEN
    MbJogExec := FALSE; jStep := 0;
ELSE
    CASE jStep OF
        0: // arm on held button (exactly one direction)
            IF JogPlus XOR JogMinus THEN
                IF JogPlus THEN MbJogVal := 16#4001; ELSE MbJogVal := 16#4002; END_IF
                MbJogExec := TRUE; tonJog(IN := FALSE); jStep := 1;
            END_IF
        1: // wait transport ack, then gap-and-repeat while still held
            tonJog(IN := TRUE, PT := T#500MS);
            IF MbJogDone OR tonJog.Q THEN
                MbJogExec := FALSE; tonJog(IN := FALSE); jStep := 0;
            END_IF
    END_CASE
    IF NOT (JogPlus XOR JogMinus) THEN
        MbJogExec := FALSE; jStep := 0;
    END_IF
END_IF

// Cyclic status monitoring comes free with the 0x1003 read channel:
// bit 0x01 = drive fault (in addition to the ALM DI). Diagnostic only.

END_FUNCTION_BLOCK

// Device/Application/03_L2_Mechanisms/FB_Press
(* ============================================================
   FB_Press — one clamshell press. Wraps FB_PressDrive (paths:
   0=OPEN 1=SMASH 2=HOLD). Executes the force/position profile:
   CLOSE->SMASH (smashDurS) -> BACK OFF to HOLD (light contact)
   -> stays HOLDING until MCMD_OPEN. Product-quality decision:
   never full force for the whole cook. Runs in T_App.
   Commands: MCMD_HOME(=open), MCMD_PROFILE, MCMD_OPEN.
   ============================================================ *)
FUNCTION_BLOCK FB_Press
VAR_INPUT
    Enable  : BOOL;
    Cmd     : ST_MechCmd;
    CmdExec : BOOL;
    Abort   : BOOL;
    Sim     : BOOL;
    PressId : INT;
    Recipe  : ST_Recipe;
    CycleMs : LREAL := 20.0;
END_VAR
VAR_IN_OUT
    Drv : FB_PressDrive;
END_VAR
VAR_OUTPUT
    Busy, Done, Error : BOOL;
    ErrorID : UDINT;
    State   : UINT;
    IsOpen  : BOOL;
    Holding : BOOL;
    DwellS  : LREAL;     // time at smash+hold, for HACCP
END_VAR
VAR
    iSt     : INT;
    rtExec : R_TRIG;
    smashT : LREAL;
    scale  : LREAL;
    tonTO  : TON;        // watchdog: any Busy state stuck -> labeled timeout
END_VAR


rtExec(CLK := CmdExec);
scale := 1.0;
IF Sim THEN scale := GVL_Cfg.SIM_TIME_SCALE; END_IF

IF Abort THEN
    iSt := 0; Busy := FALSE;
    Drv.PathExec := FALSE; Drv.WriteParams := FALSE; Drv.HomeExec := FALSE;
END_IF
IF Drv.Error AND (iSt <> 0) THEN
    iSt := 0; Busy := FALSE; Error := TRUE; ErrorID := Drv.ErrorID;
    Drv.PathExec := FALSE; Drv.WriteParams := FALSE; Drv.HomeExec := FALSE;
END_IF

// watchdog — Busy states only (HOLDING has Busy=FALSE, so a long cook never trips it)
tonTO(IN := Busy, PT := GVL_Cfg.TO_MECH);
IF tonTO.Q AND Busy THEN
    iSt := 0; Busy := FALSE; Error := TRUE;
    ErrorID := F_Err(GVL_Cfg.SS_PRESS_0 + TO_UINT(PressId), GVL_Cfg.ERR_TIMEOUT);
    Drv.PathExec := FALSE; Drv.WriteParams := FALSE;
END_IF

CASE iSt OF
    0: // idle
        IF Enable AND rtExec.Q THEN
            Done := FALSE; Error := FALSE; ErrorID := 0;
            IF (Cmd.code = GVL_Cfg.MCMD_PROFILE) THEN
                IF NOT IsOpen THEN
                    Error := TRUE; ErrorID := F_Err(GVL_Cfg.SS_PRESS_0 + TO_UINT(PressId), GVL_Cfg.ERR_INTERLOCK);
                ELSE
                    DwellS := 0.0; smashT := 0.0;
                    // push PR positions (recipe + per-press calibration trim)
                    // to the drive before commanding motion
                    Drv.OpenPosMm  := GVL_Cfg.PRESS_OPEN_MM;
                    Drv.SmashPosMm := Recipe.smashPosMm + GVL_Par.pressTrimMm[PressId];
                    Drv.HoldPosMm  := Recipe.holdPosMm  + GVL_Par.pressTrimMm[PressId];
                    Drv.WriteParams := TRUE;
                    iSt := 5; Busy := TRUE; IsOpen := FALSE;
                END_IF
            ELSIF (Cmd.code = GVL_Cfg.MCMD_OPEN) THEN
                Drv.PathNo := 0; Drv.PathExec := TRUE;          // OPEN
                iSt := 30; Busy := TRUE; Holding := FALSE;
            ELSIF (Cmd.code = GVL_Cfg.MCMD_HOME) THEN
                Drv.HomeExec := TRUE;                           // re-reference, then open
                iSt := 40; Busy := TRUE; Holding := FALSE;
            ELSE
                Error := TRUE; ErrorID := F_Err(GVL_Cfg.SS_PRESS_0 + TO_UINT(PressId), GVL_Cfg.ERR_BAD_CMD);
            END_IF
        END_IF
    5: // wait for PR table confirmed in drive, then smash
        IF Drv.ParamsValid THEN
            Drv.WriteParams := FALSE;
            Drv.PathNo := 1; Drv.PathExec := TRUE;              // SMASH
            iSt := 10;
        ELSIF Drv.ParamErr THEN
            Drv.WriteParams := FALSE;
            iSt := 0; Busy := FALSE; Error := TRUE;
            ErrorID := F_Err(GVL_Cfg.SS_PRESS_0 + TO_UINT(PressId), GVL_Cfg.ERR_DRIVE);
        END_IF
    10: // closing to smash position
        IF Drv.Done THEN
            Drv.PathExec := FALSE; iSt := 11;
        END_IF
    11: // dwell at smash force/position
        smashT := smashT + CycleMs / 1000.0 * scale;
        DwellS := DwellS + CycleMs / 1000.0 * scale;
        IF smashT >= Recipe.smashDurS THEN
            Drv.PathNo := 2; Drv.PathExec := TRUE;              // BACK OFF -> HOLD
            iSt := 12;
        END_IF
    12:
        IF Drv.Done THEN
            Drv.PathExec := FALSE;
            iSt := 20; Busy := FALSE; Done := TRUE; Holding := TRUE;
        END_IF
    20: // HOLDING for cook duration (open on command)
        DwellS := DwellS + CycleMs / 1000.0 * scale;
        IF Enable AND rtExec.Q AND (Cmd.code = GVL_Cfg.MCMD_OPEN) THEN
            Done := FALSE;
            Drv.PathNo := 0; Drv.PathExec := TRUE;
            iSt := 30; Busy := TRUE; Holding := FALSE;
        END_IF
    30: // opening
        IF Drv.Done THEN
            Drv.PathExec := FALSE;
            iSt := 0; Busy := FALSE; Done := TRUE; IsOpen := TRUE;
        END_IF
    40: // homing the drive (MCMD_HOME); when referenced, open
        IF Drv.Homed AND NOT Drv.HomeBusy THEN
            Drv.HomeExec := FALSE;
            Drv.PathNo := 0; Drv.PathExec := TRUE;              // then OPEN
            iSt := 30;
        END_IF
END_CASE
State := TO_UINT(iSt);

END_FUNCTION_BLOCK

// Device/Application/02_L1_Drivers/FB_SensorIn
(* ============================================================
   FB_SensorIn — debounced digital input.
   SIM: output follows SimValue directly.
   ============================================================ *)
FUNCTION_BLOCK FB_SensorIn
VAR_INPUT
    Sim        : BOOL;
    SimValue   : BOOL;
    iRaw       : BOOL;
    DebounceMs : LREAL := 40.0;
    CycleMs    : LREAL := 20.0;
END_VAR
VAR_OUTPUT
    Q : BOOL;
END_VAR
VAR
    acc : LREAL;
    lastRaw : BOOL;
END_VAR

IF Sim THEN
    Q := SimValue;
ELSE
    IF iRaw = lastRaw THEN
        acc := acc + CycleMs;
        IF acc >= DebounceMs THEN Q := iRaw; END_IF
    ELSE
        acc := 0.0;
        lastRaw := iRaw;
    END_IF
END_IF

END_FUNCTION_BLOCK

// Device/Application/02_L1_Drivers/FB_VfdIndex
(* ============================================================
   FB_VfdIndex — carousel indexing: VFD run/dir + encoder + pin.
   Pin actuator is external (FB_PneuActuator); this FB commands it
   via PinCmd and reads PinExtended/PinRetracted.
   Sequence: retract pin -> rotate (fast->creep) -> stop in window
   -> extend pin -> verify pin + encoder plausibility.
   Runs in T_App. SIM: integrates encoder; home prox modeled.
   ============================================================ *)
FUNCTION_BLOCK FB_VfdIndex
VAR_INPUT
    Sim          : BOOL;
    SubsysId     : UINT;
    Enable       : BOOL;
    HomeExec     : BOOL;
    GotoExec     : BOOL;
    TargetStation: INT;
    Bidirectional: BOOL;
    Abort        : BOOL;
    iEnc         : DINT;
    iHomeProx    : BOOL;
    PinExtended  : BOOL;
    PinRetracted : BOOL;
    CycleMs      : LREAL := 20.0;
END_VAR
VAR_OUTPUT
    qFwd, qRev  : BOOL;
    qSpeed      : INT;
    PinCmd      : BOOL := TRUE;     // TRUE = extend (locked at rest)
    ActStation  : INT := -1;
    Homed       : BOOL;
    Busy, Done, Error : BOOL;
    ErrorID     : UDINT;
END_VAR
VAR
    state      : INT;
    rtHome, rtGoto : R_TRIG;
    tonTO      : TON;
    encEff     : DINT;
    homeEff    : BOOL;
    encZero    : DINT;              // count value at station 0
    tgtCounts  : DINT;
    diff       : DINT;
    cps        : DINT;              // counts per station
    fwdDir     : BOOL;
    goingHome  : BOOL;
    simEnc     : DINT;
    stepC      : DINT;
END_VAR

cps := GVL_Cfg.ENC_CPR / TO_DINT(GVL_Cfg.STATIONS);
rtHome(CLK := HomeExec);
rtGoto(CLK := GotoExec);

// ------- feedback source -------
IF Sim THEN
    IF qFwd THEN
        stepC := TO_DINT(TO_LREAL(qSpeed) * CycleMs / 20.0);
        simEnc := simEnc + MAX(stepC, 1);
    ELSIF qRev THEN
        stepC := TO_DINT(TO_LREAL(qSpeed) * CycleMs / 20.0);
        simEnc := simEnc - MAX(stepC, 1);
    END_IF
    encEff  := simEnc;
    homeEff := ((simEnc MOD GVL_Cfg.ENC_CPR) + GVL_Cfg.ENC_CPR) MOD GVL_Cfg.ENC_CPR < 60;
ELSE
    encEff  := iEnc;
    homeEff := iHomeProx;
END_IF

IF Abort THEN
    qFwd := FALSE; qRev := FALSE; qSpeed := 0;
    state := 0; Busy := FALSE; tonTO(IN := FALSE);
END_IF

CASE state OF
    0: // idle (pin extended = locked)
        qFwd := FALSE; qRev := FALSE; qSpeed := 0;
        IF Enable AND rtHome.Q THEN
            goingHome := TRUE; state := 10; Busy := TRUE; Done := FALSE;
        ELSIF Enable AND Homed AND rtGoto.Q THEN
            IF (TargetStation < 0) OR (TargetStation >= GVL_Cfg.STATIONS) THEN
                Error := TRUE; ErrorID := F_Err(SubsysId, GVL_Cfg.ERR_BAD_CMD);
            ELSIF TargetStation = ActStation THEN
                Done := TRUE;
            ELSE
                goingHome := FALSE; state := 10; Busy := TRUE; Done := FALSE;
            END_IF
        END_IF

    10: // retract pin
        PinCmd := FALSE;
        tonTO(IN := TRUE, PT := GVL_Cfg.TO_PNEU);
        IF PinRetracted THEN
            tonTO(IN := FALSE); state := 20;
        ELSIF tonTO.Q THEN
            state := 90; ErrorID := F_Err(SubsysId, GVL_Cfg.ERR_PIN);
        END_IF

    20: // rotate
        IF goingHome THEN
            qFwd := TRUE; qSpeed := GVL_Cfg.IDX_SPEED_CREEP;
            tonTO(IN := TRUE, PT := GVL_Cfg.TO_INDEX);
            IF homeEff THEN
                qFwd := FALSE; qSpeed := 0;
                encZero := encEff;
                tonTO(IN := FALSE); state := 30;
            ELSIF tonTO.Q THEN
                state := 90; ErrorID := F_Err(SubsysId, GVL_Cfg.ERR_TIMEOUT);
            END_IF
        ELSE
            tgtCounts := encZero + TO_DINT(TargetStation) * cps;
            diff := tgtCounts - encEff;
            IF Bidirectional THEN
                // shortest signed path within one revolution
                diff := ((diff MOD GVL_Cfg.ENC_CPR) + GVL_Cfg.ENC_CPR) MOD GVL_Cfg.ENC_CPR;
                IF diff > GVL_Cfg.ENC_CPR / 2 THEN diff := diff - GVL_Cfg.ENC_CPR; END_IF
            ELSE
                diff := ((diff MOD GVL_Cfg.ENC_CPR) + GVL_Cfg.ENC_CPR) MOD GVL_Cfg.ENC_CPR;
            END_IF
            fwdDir := diff >= 0;
            qFwd := fwdDir AND (ABS(diff) > GVL_Cfg.IDX_STOP_WIN);
            qRev := (NOT fwdDir) AND (ABS(diff) > GVL_Cfg.IDX_STOP_WIN);
            IF ABS(diff) > GVL_Cfg.IDX_DECEL_WIN THEN
                qSpeed := GVL_Cfg.IDX_SPEED_FAST;
            ELSE
                qSpeed := GVL_Cfg.IDX_SPEED_CREEP;
            END_IF
            tonTO(IN := TRUE, PT := GVL_Cfg.TO_INDEX);
            IF ABS(diff) <= GVL_Cfg.IDX_STOP_WIN THEN
                qFwd := FALSE; qRev := FALSE; qSpeed := 0;
                tonTO(IN := FALSE); state := 30;
            ELSIF tonTO.Q THEN
                state := 90; ErrorID := F_Err(SubsysId, GVL_Cfg.ERR_TIMEOUT);
            END_IF
        END_IF

    30: // extend pin + verify
        PinCmd := TRUE;
        tonTO(IN := TRUE, PT := GVL_Cfg.TO_PNEU);
        IF PinExtended THEN
            tonTO(IN := FALSE);
            IF goingHome THEN
                Homed := TRUE; ActStation := 0;
            ELSE
                // encoder-vs-pin plausibility
                diff := (((encEff - encZero) MOD GVL_Cfg.ENC_CPR) + GVL_Cfg.ENC_CPR) MOD GVL_Cfg.ENC_CPR;
                IF ABS(diff - TO_DINT(TargetStation) * cps) > GVL_Cfg.IDX_VERIFY_WIN THEN
                    state := 90; ErrorID := F_Err(SubsysId, GVL_Cfg.ERR_PIN);
                    Homed := FALSE;                    // demand re-home
                    RETURN;
                END_IF
                ActStation := TargetStation;
            END_IF
            state := 0; Busy := FALSE; Done := TRUE;
        ELSIF tonTO.Q THEN
            state := 90; ErrorID := F_Err(SubsysId, GVL_Cfg.ERR_PIN);
        END_IF

    90: // fault
        qFwd := FALSE; qRev := FALSE; qSpeed := 0;
        Busy := FALSE; Error := TRUE;
        state := 0;
END_CASE

END_FUNCTION_BLOCK

// Device/Application/03_L2_Mechanisms/FB_Airlock
(* ============================================================
   FB_Airlock — chamber gate mutual exclusion. Requests are
   LEVELS; the FB grants at most one open door, closing the other
   first. ChamberSealed = both confirmed closed. Runs in T_App.
   DoorFridge = fridge-side gate, DoorChamber = griddle-side gate.
   ============================================================ *)
FUNCTION_BLOCK FB_Airlock
VAR_INPUT
    Enable         : BOOL;
    ReqFridgeOpen  : BOOL;
    ReqChamberOpen : BOOL;
    Abort          : BOOL;
END_VAR
VAR_IN_OUT
    DoorFridge  : FB_PneuActuator;
    DoorChamber : FB_PneuActuator;
END_VAR
VAR_OUTPUT
    FridgeOpen    : BOOL;
    ChamberOpen   : BOOL;
    ChamberSealed : BOOL;
    Busy, Error   : BOOL;
    ErrorID       : UDINT;
END_VAR
VAR
    wantF, wantC : BOOL;
END_VAR

wantF := Enable AND ReqFridgeOpen AND NOT Abort;
wantC := Enable AND ReqChamberOpen AND NOT Abort;

// mutual exclusion: fridge side has priority; never open one until
// the other is CONFIRMED retracted (closed)
IF wantF AND wantC THEN wantC := FALSE; END_IF
DoorFridge.Cmd  := wantF AND DoorChamber.Retracted;
DoorChamber.Cmd := wantC AND DoorFridge.Retracted;

FridgeOpen    := DoorFridge.Extended;
ChamberOpen   := DoorChamber.Extended;
ChamberSealed := DoorFridge.Retracted AND DoorChamber.Retracted;
Busy := (wantF AND NOT FridgeOpen) OR (wantC AND NOT ChamberOpen)
     OR ((NOT wantF) AND NOT DoorFridge.Retracted)
     OR ((NOT wantC) AND NOT DoorChamber.Retracted);

IF DoorFridge.Error OR DoorChamber.Error THEN
    Error := TRUE;
    ErrorID := F_Err(GVL_Cfg.SS_AIRLOCK, GVL_Cfg.ERR_TIMEOUT);
ELSE
    Error := FALSE; ErrorID := 0;
END_IF

// hard invariant — must never trip, in sim or real
IF FridgeOpen AND ChamberOpen THEN
    Error := TRUE;
    ErrorID := F_Err(GVL_Cfg.SS_AIRLOCK, GVL_Cfg.ERR_INTERLOCK);
END_IF

END_FUNCTION_BLOCK

// Device/Application/03_L2_Mechanisms/FB_Fork
(* ============================================================
   FB_Fork — tray fetch/return, 2 axes + fail-safe brake.
   Commands: MCMD_HOME, MCMD_FETCH(p1=level), MCMD_RETURN(p1=level).
   Fetch: Z to level -> tele out -> micro-lift (release stacking
   lock) -> tele in (tray drawn into chamber).
   Return: Z to level+micro -> tele out -> micro-drop (re-engage
   lock) -> tele in.
   Brake: qBrakeRelease TRUE only while Z powered & healthy; a
   feedback mismatch is MACHINE_STOP class. Runs in T_Motion.
   ============================================================ *)
FUNCTION_BLOCK FB_Fork
VAR_INPUT
    Enable  : BOOL;
    Cmd     : ST_MechCmd;
    CmdExec : BOOL;
    Abort   : BOOL;
    Sim     : BOOL;
    iBrakeOk : BOOL;
    iTrayPresent : BOOL;
END_VAR
VAR_IN_OUT
    AxZ : FB_AxisCtrl;
    AxT : FB_AxisCtrl;    // telescope
END_VAR
VAR_OUTPUT
    qBrakeRelease : BOOL;
    TrayHeld : BOOL;
    Busy, Done, Error : BOOL;
    ErrorID : UDINT;
    State : UINT;
    Homed : BOOL;
END_VAR
VAR
    iSt : INT;
    rtExec : R_TRIG;
    level : INT;
    zBase : LREAL;
    fetching : BOOL;
    brakeChk : TON;
    tonTO : TON;
    trayEff : BOOL;
END_VAR

rtExec(CLK := CmdExec);
trayEff := (Sim AND TrayHeld) OR ((NOT Sim) AND iTrayPresent);

// brake proving: release demand vs feedback
qBrakeRelease := Enable AND AxZ.Sts.powered AND NOT Abort AND NOT Error;
brakeChk(IN := (NOT Sim) AND (qBrakeRelease <> iBrakeOk), PT := T#500MS);
IF brakeChk.Q THEN
    Error := TRUE;
    ErrorID := F_Err(GVL_Cfg.SS_FORK_Z, GVL_Cfg.ERR_DRIVE);   // MACHINE_STOP via PRG_Alarms map
END_IF

IF Abort THEN
    iSt := 0; Busy := FALSE;
    AxZ.MoveExec := FALSE; AxT.MoveExec := FALSE;
    AxZ.HomeExec := FALSE; AxT.HomeExec := FALSE;
END_IF
Homed := AxZ.Sts.homed AND AxT.Sts.homed;

tonTO(IN := Busy, PT := GVL_Cfg.TO_MECH);
IF tonTO.Q AND Busy THEN
    iSt := 0; Busy := FALSE; Error := TRUE;
    ErrorID := F_Err(GVL_Cfg.SS_FORK, GVL_Cfg.ERR_TIMEOUT);
END_IF

CASE iSt OF
    0:
        IF Enable AND rtExec.Q AND NOT Error THEN
            Done := FALSE; ErrorID := 0;
            CASE Cmd.code OF
                1:  (* MCMD_HOME *)  iSt := 10; Busy := TRUE;
                20, 21: (* MCMD_FETCH / MCMD_RETURN *)
                    level := TO_INT(Cmd.p1);
                    IF (level < 0) OR (level >= GVL_Cfg.TRAY_LEVELS) THEN
                        Error := TRUE; ErrorID := F_Err(GVL_Cfg.SS_FORK, GVL_Cfg.ERR_BAD_CMD);
                    ELSE
                        fetching := (Cmd.code = GVL_Cfg.MCMD_FETCH);  // constant compare OK outside CASE labels
                        zBase := GVL_Cfg.FORK_Z0 + TO_LREAL(level) * GVL_Cfg.FORK_LEVEL_H;
                        iSt := 20; Busy := TRUE;
                    END_IF
            ELSE
                Error := TRUE; ErrorID := F_Err(GVL_Cfg.SS_FORK, GVL_Cfg.ERR_BAD_CMD);
            END_CASE
        END_IF
    10: // HOME: telescope retract first, then Z
        AxT.HomeExec := TRUE;
        IF AxT.Sts.homed THEN AxT.HomeExec := FALSE; iSt := 11; END_IF
    11:
        AxZ.HomeExec := TRUE;
        IF AxZ.Sts.homed THEN
            AxZ.HomeExec := FALSE; iSt := 0; Busy := FALSE; Done := TRUE;
        END_IF
    20: // Z to level (fetch: exact; return: +microlift so tray clears)
        IF fetching THEN AxZ.TargetPos := zBase;
        ELSE AxZ.TargetPos := zBase + GVL_Cfg.FORK_MICROLIFT; END_IF
        AxZ.Vel := GVL_Cfg.F_VEL; AxZ.Acc := GVL_Cfg.F_ACC;
        AxZ.MoveExec := TRUE;
        IF AxZ.Done THEN AxZ.MoveExec := FALSE; iSt := 21; END_IF
        IF AxZ.Error THEN iSt := 90; END_IF
    21: // telescope out
        AxT.TargetPos := GVL_Cfg.FORK_TELE_OUT; AxT.Vel := GVL_Cfg.F_VEL; AxT.Acc := GVL_Cfg.F_ACC;
        AxT.MoveExec := TRUE;
        IF AxT.Done THEN AxT.MoveExec := FALSE; iSt := 22; END_IF
        IF AxT.Error THEN iSt := 90; END_IF
    22: // micro-lift (fetch) or micro-drop (return)
        IF fetching THEN AxZ.TargetPos := zBase + GVL_Cfg.FORK_MICROLIFT;
        ELSE AxZ.TargetPos := zBase; END_IF
        AxZ.MoveExec := TRUE;
        IF AxZ.Done THEN AxZ.MoveExec := FALSE; iSt := 23; END_IF
        IF AxZ.Error THEN iSt := 90; END_IF
    23: // telescope in
        AxT.TargetPos := GVL_Cfg.FORK_TELE_IN; AxT.MoveExec := TRUE;
        IF AxT.Done THEN
            AxT.MoveExec := FALSE;
            IF fetching THEN
                TrayHeld := TRUE;
                IF Sim OR trayEff THEN
                    iSt := 0; Busy := FALSE; Done := TRUE;
                ELSE
                    TrayHeld := FALSE;
                    iSt := 0; Busy := FALSE; Error := TRUE;
                    ErrorID := F_Err(GVL_Cfg.SS_FORK, GVL_Cfg.ERR_SENSOR);  // tray not present
                END_IF
            ELSE
                TrayHeld := FALSE;
                iSt := 0; Busy := FALSE; Done := TRUE;
            END_IF
        END_IF
        IF AxT.Error THEN iSt := 90; END_IF
    90:
        AxZ.MoveExec := FALSE; AxT.MoveExec := FALSE;
        IF ErrorID = 0 THEN
            IF AxZ.Error THEN ErrorID := AxZ.ErrorID;
            ELSIF AxT.Error THEN ErrorID := AxT.ErrorID;
            ELSE ErrorID := F_Err(GVL_Cfg.SS_FORK, GVL_Cfg.ERR_DRIVE); END_IF
        END_IF
        iSt := 0; Busy := FALSE; Error := TRUE;
END_CASE
State := TO_UINT(iSt);

END_FUNCTION_BLOCK

// Device/Application/03_L2_Mechanisms/FB_FridgeCarousel
(* ============================================================
   FB_FridgeCarousel — tray column indexing (2 faces). Identical
   pattern to the griddle carousel, no rotation permissive beyond
   fork-retracted (wired by caller as Permissive). Unidirectional
   is acceptable here. Runs in T_App.
   ============================================================ *)
FUNCTION_BLOCK FB_FridgeCarousel
VAR_INPUT
    Enable     : BOOL;
    HomeExec   : BOOL;
    GotoExec   : BOOL;
    TargetFace : INT;       // 0..1 mapped to stations 0 / STATIONS/2
    Permissive : BOOL;      // fork telescope retracted
    Abort      : BOOL;
END_VAR
VAR_IN_OUT
    Vfd : FB_VfdIndex;
    Pin : FB_PneuActuator;
END_VAR
VAR_OUTPUT
    ActFace : INT;
    Homed   : BOOL;
    Busy, Done, Error : BOOL;
    ErrorID : UDINT;
END_VAR
VAR
    rtGoto : R_TRIG;
END_VAR

rtGoto(CLK := GotoExec);
IF rtGoto.Q AND NOT Permissive THEN
    Error := TRUE;
    ErrorID := F_Err(GVL_Cfg.SS_FRIDGE_CAR, GVL_Cfg.ERR_INTERLOCK);
END_IF

Pin.Cmd          := Vfd.PinCmd;
Vfd.PinExtended  := Pin.Extended;
Vfd.PinRetracted := Pin.Retracted;

Vfd.Enable   := Enable;
Vfd.Abort    := Abort;
Vfd.HomeExec := HomeExec;
Vfd.GotoExec := GotoExec AND Permissive;
Vfd.TargetStation := TargetFace * (GVL_Cfg.STATIONS / 2);
Vfd.Bidirectional := FALSE;

IF Vfd.ActStation = 0 THEN ActFace := 0;
ELSIF Vfd.ActStation = GVL_Cfg.STATIONS / 2 THEN ActFace := 1;
ELSE ActFace := -1; END_IF
Homed := Vfd.Homed;
Busy  := Vfd.Busy;
Done  := Vfd.Done;
IF Vfd.Error OR Pin.Error THEN
    Error := TRUE;
    IF Vfd.Error THEN ErrorID := Vfd.ErrorID; ELSE ErrorID := Pin.ErrorID; END_IF
END_IF

END_FUNCTION_BLOCK

// Device/Application/03_L2_Mechanisms/FB_Gantry
(* ============================================================
   FB_Gantry — pick/place mechanism. Standard interface (spec sec.12).
   Owns sequencing only; axis FB bodies are called in PRG_Motion.
   Commands: MCMD_HOME, MCMD_PICK(p1=trayIdx 0..23),
             MCMD_PLACE(p1=slot 0..5), MCMD_PARK, MCMD_SANITIZE.
   Coordinated XY = simultaneous X + theta targets (v1; swap to
   interpolated transform after IK validation without touching
   callers — see method note in spec 9.1).
   Runs in T_Motion.
   ============================================================ *)
FUNCTION_BLOCK FB_Gantry
VAR_INPUT
    Enable  : BOOL;
    Cmd     : ST_MechCmd;
    CmdExec : BOOL;
    Abort   : BOOL;
    Sim     : BOOL;
END_VAR
VAR_IN_OUT
    AxX  : FB_AxisCtrl;
    AxT  : FB_AxisCtrl;
    AxZ  : FB_AxisCtrl;
    Grip : FB_Gripper;
    IK   : FB_IKTransform;
END_VAR
VAR_OUTPUT
    Busy, Done, Error : BOOL;
    ErrorID : UDINT;
    State   : UINT;
    Homed   : BOOL;
    Parked  : BOOL;
END_VAR
VAR
    iSt      : INT;
    rtExec  : R_TRIG;
    cmdL    : ST_MechCmd;
    tgtX, tgtY : LREAL;
    zTarget : LREAL;
    idx, row, col : INT;
    tonTO   : TON;
END_VAR


rtExec(CLK := CmdExec);

IF Abort THEN
    iSt := 0; Busy := FALSE;
    AxX.MoveExec := FALSE; AxT.MoveExec := FALSE; AxZ.MoveExec := FALSE;
    AxX.HomeExec := FALSE; AxT.HomeExec := FALSE; AxZ.HomeExec := FALSE;
    tonTO(IN := FALSE);
END_IF

Homed  := AxX.Sts.homed AND AxT.Sts.homed AND AxZ.Sts.homed;
Parked := Homed AND (iSt = 0) AND (ABS(AxX.Sts.actPos - GVL_Cfg.GX_PARK) < 2.0);

tonTO(IN := Busy, PT := GVL_Cfg.TO_MECH);
IF tonTO.Q AND Busy THEN
    iSt := 0; Busy := FALSE; Error := TRUE;
    ErrorID := F_Err(GVL_Cfg.SS_GANTRY, GVL_Cfg.ERR_TIMEOUT);
END_IF

CASE iSt OF
    0: // IDLE — accept command
        IF Enable AND rtExec.Q THEN
            cmdL := Cmd; Done := FALSE; Error := FALSE; ErrorID := 0;
            CASE cmdL.code OF
                1:  (* MCMD_HOME *)     iSt := 10; Busy := TRUE;
                10: (* MCMD_PICK *)
                    idx := TO_INT(cmdL.p1);
                    row := idx / GVL_Cfg.TRAY_COLS;  col := idx MOD GVL_Cfg.TRAY_COLS;
                    tgtX := GVL_Cfg.PICK_BASE_X + TO_LREAL(col) * GVL_Cfg.PICK_SPACING_X + GVL_Par.pickOffsetX;
                    tgtY := GVL_Cfg.PICK_BASE_Y + TO_LREAL(row) * GVL_Cfg.PICK_SPACING_Y + GVL_Par.pickOffsetY;
                    zTarget := GVL_Cfg.GZ_PICK;
                    iSt := 20; Busy := TRUE;
                11: (* MCMD_PLACE *)
                    idx := TO_INT(cmdL.p1);
                    row := idx / GVL_Cfg.PLACE_COLS; col := idx MOD GVL_Cfg.PLACE_COLS;
                    tgtX := GVL_Cfg.PLACE_BASE_X + TO_LREAL(col) * GVL_Cfg.PLACE_SPC_X + GVL_Par.placeOffsetX;
                    tgtY := GVL_Cfg.PLACE_BASE_Y + TO_LREAL(row) * GVL_Cfg.PLACE_SPC_Y + GVL_Par.placeOffsetY;
                    zTarget := GVL_Cfg.GZ_PLACE;
                    iSt := 20; Busy := TRUE;
                2:  (* MCMD_PARK *)
                    tgtX := GVL_Cfg.GX_PARK; tgtY := GVL_Cfg.ARM_LEN * 0.0;
                    iSt := 60; Busy := TRUE;
                13: (* MCMD_SANITIZE *)
                    tgtX := GVL_Cfg.GX_MAX;  tgtY := 0.0;    // wash-station pose TODO
                    iSt := 60; Busy := TRUE;
            ELSE
                Error := TRUE; ErrorID := F_Err(GVL_Cfg.SS_GANTRY, GVL_Cfg.ERR_BAD_CMD);
            END_CASE
        END_IF

    10: // HOME: Z up first, then theta safe, then X (collision-safe)
        AxZ.HomeExec := TRUE;
        IF AxZ.Sts.homed THEN AxZ.HomeExec := FALSE; iSt := 11; END_IF
    11:
        AxT.HomeExec := TRUE;
        IF AxT.Sts.homed THEN AxT.HomeExec := FALSE; iSt := 12; END_IF
    12:
        AxX.HomeExec := TRUE;
        IF AxX.Sts.homed THEN
            AxX.HomeExec := FALSE;
            iSt := 0; Busy := FALSE; Done := TRUE;
        END_IF

    20: // PICK/PLACE step 1: Z up
        AxZ.TargetPos := GVL_Cfg.GZ_UP;
        AxZ.Vel := GVL_Cfg.Z_VEL; AxZ.Acc := GVL_Cfg.Z_ACC;
        AxZ.MoveExec := TRUE;
        IF AxZ.Done THEN AxZ.MoveExec := FALSE; iSt := 21; END_IF
        IF AxZ.Error THEN iSt := 90; END_IF
    21: // step 2: IK + coordinated XY
        IK(xCart := tgtX, yCart := tgtY);
        IF NOT IK.Reachable THEN
            iSt := 0; Busy := FALSE; Error := TRUE;
            ErrorID := F_Err(GVL_Cfg.SS_GANTRY, GVL_Cfg.ERR_UNREACH);
        ELSE
            AxX.TargetPos := IK.xLin;     AxX.Vel := GVL_Cfg.G_VEL; AxX.Acc := GVL_Cfg.G_ACC;
            AxT.TargetPos := IK.thetaDeg; AxT.Vel := GVL_Cfg.T_VEL; AxT.Acc := GVL_Cfg.T_ACC;
            AxX.MoveExec := TRUE; AxT.MoveExec := TRUE;
            iSt := 22;
        END_IF
    22:
        IF AxX.Done AND AxT.Done THEN
            AxX.MoveExec := FALSE; AxT.MoveExec := FALSE; iSt := 23;
        END_IF
        IF AxX.Error OR AxT.Error THEN iSt := 90; END_IF
    23: // step 3: Z dip
        AxZ.TargetPos := zTarget; AxZ.MoveExec := TRUE;
        IF AxZ.Done THEN AxZ.MoveExec := FALSE; iSt := 24; END_IF
        IF AxZ.Error THEN iSt := 90; END_IF
    24: // step 4: arm grip/release; result checked next scan (Grip.Done may be stale this scan)
        IF cmdL.code = GVL_Cfg.MCMD_PICK THEN
            Grip.AcquireExec := TRUE;
        ELSE
            Grip.ReleaseExec := TRUE;
        END_IF
        iSt := 26;
    26: // wait gripper result
        IF Grip.Done THEN
            Grip.AcquireExec := FALSE; Grip.ReleaseExec := FALSE; iSt := 25;
        END_IF
        IF Grip.Error THEN
            Grip.AcquireExec := FALSE; Grip.ReleaseExec := FALSE;
            ErrorID := Grip.ErrorID; iSt := 90;
        END_IF
    25: // step 5: Z up -> done
        AxZ.TargetPos := GVL_Cfg.GZ_UP; AxZ.MoveExec := TRUE;
        IF AxZ.Done THEN
            AxZ.MoveExec := FALSE;
            iSt := 0; Busy := FALSE; Done := TRUE;
        END_IF
        IF AxZ.Error THEN iSt := 90; END_IF

    60: // PARK / SANITIZE: Z up then XY
        AxZ.TargetPos := GVL_Cfg.GZ_UP; AxZ.MoveExec := TRUE;
        IF AxZ.Done THEN AxZ.MoveExec := FALSE; iSt := 61; END_IF
        IF AxZ.Error THEN iSt := 90; END_IF
    61:
        IK(xCart := tgtX + GVL_Cfg.ARM_LEN, yCart := tgtY);  // park pose: arm at 0 deg
        AxX.TargetPos := tgtX;  AxX.Vel := GVL_Cfg.G_VEL; AxX.Acc := GVL_Cfg.G_ACC;
        AxT.TargetPos := 0.0;   AxT.Vel := GVL_Cfg.T_VEL; AxT.Acc := GVL_Cfg.T_ACC;
        AxX.MoveExec := TRUE; AxT.MoveExec := TRUE;
        iSt := 62;
    62:
        IF AxX.Done AND AxT.Done THEN
            AxX.MoveExec := FALSE; AxT.MoveExec := FALSE;
            iSt := 0; Busy := FALSE; Done := TRUE;
        END_IF
        IF AxX.Error OR AxT.Error THEN iSt := 90; END_IF

    90: // fault funnel
        AxX.MoveExec := FALSE; AxT.MoveExec := FALSE; AxZ.MoveExec := FALSE;
        Grip.AcquireExec := FALSE; Grip.ReleaseExec := FALSE;
        IF ErrorID = 0 THEN
            IF AxX.Error THEN ErrorID := AxX.ErrorID;
            ELSIF AxT.Error THEN ErrorID := AxT.ErrorID;
            ELSIF AxZ.Error THEN ErrorID := AxZ.ErrorID;
            ELSE ErrorID := F_Err(GVL_Cfg.SS_GANTRY, GVL_Cfg.ERR_DRIVE); END_IF
        END_IF
        iSt := 0; Busy := FALSE; Error := TRUE;
END_CASE
State := TO_UINT(iSt);

END_FUNCTION_BLOCK

// Device/Application/03_L2_Mechanisms/FB_Gripper
(* ============================================================
   FB_Gripper — v1 stub over one pneumatic channel. INTERFACE IS
   FROZEN: swap internals when the real effector is designed.
   Owned pneu FB instance is external (GVL_Mech.fbPneuGrip), body
   called in PRG_Carousels; this FB only writes Cmd / reads status.
   Runs in T_Motion (with FB_Gantry).
   ============================================================ *)
FUNCTION_BLOCK FB_Gripper
VAR_INPUT
    Sim         : BOOL;
    AcquireExec : BOOL;    // edge
    ReleaseExec : BOOL;
    iAcquired   : BOOL;    // patty-acquired feedback (sim: modeled)
    CycleMs     : LREAL := 4.0;
END_VAR
VAR_IN_OUT
    Pneu : FB_PneuActuator;
END_VAR
VAR_OUTPUT
    Holding : BOOL;
    Busy, Done, Error : BOOL;
    ErrorID : UDINT;
END_VAR
VAR
    state : INT;
    rtA, rtR : R_TRIG;
    tonTO : TON;
    acqEff : BOOL;
END_VAR

rtA(CLK := AcquireExec);
rtR(CLK := ReleaseExec);
acqEff := (Sim AND Pneu.Extended) OR ((NOT Sim) AND iAcquired);

CASE state OF
    0:
        IF rtA.Q THEN Pneu.Cmd := TRUE;  state := 1; Busy := TRUE; Done := FALSE; tonTO(IN := FALSE); END_IF
        IF rtR.Q THEN Pneu.Cmd := FALSE; state := 2; Busy := TRUE; Done := FALSE; tonTO(IN := FALSE); END_IF
    1: // acquiring
        tonTO(IN := TRUE, PT := GVL_Cfg.TO_PNEU);
        IF Pneu.Extended AND acqEff THEN
            Holding := TRUE; state := 0; Busy := FALSE; Done := TRUE;
        ELSIF tonTO.Q THEN
            state := 0; Busy := FALSE; Error := TRUE;
            ErrorID := F_Err(GVL_Cfg.SS_GRIPPER, GVL_Cfg.ERR_TIMEOUT);
        END_IF
    2: // releasing
        tonTO(IN := TRUE, PT := GVL_Cfg.TO_PNEU);
        IF Pneu.Retracted THEN
            Holding := FALSE; state := 0; Busy := FALSE; Done := TRUE;
        ELSIF tonTO.Q THEN
            state := 0; Busy := FALSE; Error := TRUE;
            ErrorID := F_Err(GVL_Cfg.SS_GRIPPER, GVL_Cfg.ERR_TIMEOUT);
        END_IF
END_CASE

END_FUNCTION_BLOCK

// Device/Application/03_L2_Mechanisms/FB_IKTransform
(* ============================================================
   FB_IKTransform — Cartesian (x,y) -> gantry (xLinear, thetaDeg).
   Model: carriage travels along X at y=0; arm of length ARM_LEN
   pivots on carriage:  x = xLin + L*cos(theta),  y = L*sin(theta)
   Solution: theta = ASIN(y/L) (elbow toward +x), xLin = x - L*cos.
   MILESTONE M1 GATE: validate over the full tray+griddle table in
   simulation (see TESTING_GUIDE TC-02) before any hardware motion.
   ============================================================ *)
FUNCTION_BLOCK FB_IKTransform
VAR_INPUT
    xCart : LREAL;
    yCart : LREAL;
END_VAR
VAR_OUTPUT
    xLin      : LREAL;
    thetaDeg  : LREAL;
    Reachable : BOOL;
END_VAR
VAR
    rNorm      : LREAL;
    thetaR : LREAL;
    PI_    : LREAL := 3.14159265358979;
END_VAR

Reachable := FALSE;
IF ABS(yCart) > GVL_Cfg.ARM_LEN THEN RETURN; END_IF
rNorm := yCart / GVL_Cfg.ARM_LEN;
thetaR := ASIN(rNorm);
thetaDeg := thetaR * 180.0 / PI_;
xLin := xCart - GVL_Cfg.ARM_LEN * COS(thetaR);
Reachable := (xLin >= GVL_Cfg.GX_MIN) AND (xLin <= GVL_Cfg.GX_MAX)
         AND (thetaDeg >= GVL_Cfg.THETA_MIN) AND (thetaDeg <= GVL_Cfg.THETA_MAX);

END_FUNCTION_BLOCK

// Device/Application/03_L2_Mechanisms/FB_GriddleCarousel
(* ============================================================
   FB_GriddleCarousel — thin coordinator over FB_VfdIndex + pin
   FB_PneuActuator with the ROTATION PERMISSIVE interlock:
   all presses open + gantry parked + scraper parked (computed by
   PRG_JobExec, wired in PRG_Carousels).
   ActStation = index of the griddle currently AT THE LOAD STATION.
   Griddle g is at scrape station when ActStation = (g+2) MOD 4.
   Runs in T_App.
   ============================================================ *)
FUNCTION_BLOCK FB_GriddleCarousel
VAR_INPUT
    Enable        : BOOL;
    HomeExec      : BOOL;
    GotoExec      : BOOL;
    TargetStation : INT;
    RotatePermissive : BOOL;
    Abort         : BOOL;
END_VAR
VAR_IN_OUT
    Vfd : FB_VfdIndex;
    Pin : FB_PneuActuator;
END_VAR
VAR_OUTPUT
    ActStation : INT;
    Homed      : BOOL;
    Busy, Done, Error : BOOL;
    ErrorID    : UDINT;
END_VAR
VAR
    rtGoto : R_TRIG;
    blocked: BOOL;
END_VAR

rtGoto(CLK := GotoExec);

// wire pin actuator to indexing driver
Pin.Cmd          := Vfd.PinCmd;
Vfd.PinExtended  := Pin.Extended;
Vfd.PinRetracted := Pin.Retracted;

blocked := rtGoto.Q AND NOT RotatePermissive;
IF blocked THEN
    Error := TRUE;
    ErrorID := F_Err(GVL_Cfg.SS_GRID_CAR, GVL_Cfg.ERR_INTERLOCK);
END_IF

Vfd.Enable   := Enable;
Vfd.Abort    := Abort;
Vfd.HomeExec := HomeExec;
Vfd.GotoExec := GotoExec AND RotatePermissive;
Vfd.TargetStation := TargetStation;
Vfd.Bidirectional := TRUE;                 // shortest signed path

ActStation := Vfd.ActStation;
Homed := Vfd.Homed;
Busy  := Vfd.Busy;
Done  := Vfd.Done;
IF Vfd.Error THEN
    Error := TRUE; ErrorID := Vfd.ErrorID;
ELSIF NOT blocked THEN
    Error := FALSE; ErrorID := 0;
END_IF
IF Pin.Error THEN
    Error := TRUE; ErrorID := Pin.ErrorID;
END_IF

END_FUNCTION_BLOCK

// Device/Application/03_L2_Mechanisms/FB_Refrigeration
(* ============================================================
   FB_Refrigeration — compressor hysteresis + HACCP excursion
   timer. Runs in T_App. SIM: simple pulldown/heat-leak model.
   Excursion (> setpoint+0.5 C for FRIDGE_EXC_S) -> QUARANTINE
   flag (mapped by PRG_Alarms).
   ============================================================ *)
FUNCTION_BLOCK FB_Refrigeration
VAR_INPUT
    Sim      : BOOL;
    Enable   : BOOL;
    iTempRaw : INT;       // 0.1 degC
    CycleMs  : LREAL := 20.0;
END_VAR
VAR_OUTPUT
    qCompressor : BOOL;
    ActC        : LREAL;
    AtSet       : BOOL;
    Excursion   : BOOL;
    ErrorID     : UDINT;
END_VAR
VAR
    simC   : LREAL := 25.0;   // pulldown from ambient at boot
    excT   : LREAL;
    minRun : TON;
    minOff : TON;
    compReq: BOOL;
END_VAR

IF Sim THEN
    IF qCompressor THEN
        simC := simC - 0.15 * (CycleMs / 1000.0) * GVL_Cfg.SIM_TIME_SCALE;
    ELSE
        simC := simC + 0.03 * (CycleMs / 1000.0) * GVL_Cfg.SIM_TIME_SCALE;
    END_IF
    simC := LIMIT(1.0, simC, 30.0);
    ActC := simC;
ELSE
    ActC := TO_LREAL(iTempRaw) / 10.0;
END_IF

// hysteresis with min run/stop (compressor protection)
IF ActC > GVL_Cfg.FRIDGE_SET_C + GVL_Cfg.FRIDGE_HYST_C THEN compReq := TRUE; END_IF
IF ActC < GVL_Cfg.FRIDGE_SET_C - GVL_Cfg.FRIDGE_HYST_C THEN compReq := FALSE; END_IF
minRun(IN := qCompressor, PT := T#60S);
minOff(IN := NOT qCompressor, PT := T#60S);
IF Enable THEN
    IF compReq AND (minOff.Q OR Sim) THEN qCompressor := TRUE; END_IF
    IF (NOT compReq) AND (minRun.Q OR Sim) THEN qCompressor := FALSE; END_IF
ELSE
    qCompressor := FALSE;
END_IF

AtSet := ActC <= GVL_Cfg.FRIDGE_SET_C + 1.0;

IF Enable AND (ActC > GVL_Cfg.FRIDGE_SET_C + 0.5) AND AtSet = FALSE AND (GVL_Sts.mode = E_MachMode.RUN) THEN
    excT := excT + CycleMs / 1000.0 * GVL_Cfg.SIM_TIME_SCALE;
ELSE
    excT := 0.0;
END_IF
Excursion := excT >= GVL_Cfg.FRIDGE_EXC_S;
IF Excursion THEN
    ErrorID := F_Err(GVL_Cfg.SS_REFRIG, GVL_Cfg.ERR_SENSOR);
END_IF

END_FUNCTION_BLOCK

// Device/Application/03_L2_Mechanisms/FB_Scraper
(* ============================================================
   FB_Scraper — sweep mechanism. Commands: MCMD_HOME, MCMD_PARK,
   MCMD_SWEEP(p1=strokeIdx 0..2). One SWEEP = position at row,
   Z engage, X sweep across, Z up, return. Caller (JobExec)
   guarantees the interlock: griddle at scrape station, clamshell
   open, press retracted. Runs in T_Motion.
   ============================================================ *)
FUNCTION_BLOCK FB_Scraper
VAR_INPUT
    Enable  : BOOL;
    Cmd     : ST_MechCmd;
    CmdExec : BOOL;
    Abort   : BOOL;
    Sim     : BOOL;
    InterlockOk : BOOL;    // from JobExec: safe to engage
END_VAR
VAR_IN_OUT
    AxX : FB_AxisCtrl;
    AxY : FB_AxisCtrl;
    AxZ : FB_AxisCtrl;
END_VAR
VAR_OUTPUT
    Busy, Done, Error : BOOL;
    ErrorID : UDINT;
    State   : UINT;
    Homed, Parked : BOOL;
END_VAR
VAR
    iSt     : INT;
    rtExec : R_TRIG;
    stroke : INT;
    tonTO  : TON;
END_VAR

rtExec(CLK := CmdExec);
IF Abort THEN
    iSt := 0; Busy := FALSE;
    AxX.MoveExec := FALSE; AxY.MoveExec := FALSE; AxZ.MoveExec := FALSE;
    AxX.HomeExec := FALSE; AxY.HomeExec := FALSE; AxZ.HomeExec := FALSE;
END_IF
Homed  := AxX.Sts.homed AND AxY.Sts.homed AND AxZ.Sts.homed;
Parked := Homed AND (iSt = 0);

tonTO(IN := Busy, PT := GVL_Cfg.TO_MECH);
IF tonTO.Q AND Busy THEN
    iSt := 0; Busy := FALSE; Error := TRUE;
    ErrorID := F_Err(GVL_Cfg.SS_SCRAPER, GVL_Cfg.ERR_TIMEOUT);
END_IF

CASE iSt OF
    0:
        IF Enable AND rtExec.Q THEN
            Done := FALSE; Error := FALSE; ErrorID := 0;
            CASE Cmd.code OF
                1:  (* MCMD_HOME *)  iSt := 10; Busy := TRUE;
                30: (* MCMD_SWEEP *)
                    stroke := TO_INT(Cmd.p1);
                    IF (stroke < 0) OR (stroke >= GVL_Cfg.SC_STROKES) THEN
                        Error := TRUE; ErrorID := F_Err(GVL_Cfg.SS_SCRAPER, GVL_Cfg.ERR_BAD_CMD);
                    ELSIF NOT InterlockOk THEN
                        Error := TRUE; ErrorID := F_Err(GVL_Cfg.SS_SCRAPER, GVL_Cfg.ERR_INTERLOCK);
                    ELSE
                        iSt := 20; Busy := TRUE;
                    END_IF
                2:  (* MCMD_PARK *)  iSt := 60; Busy := TRUE;
            ELSE
                Error := TRUE; ErrorID := F_Err(GVL_Cfg.SS_SCRAPER, GVL_Cfg.ERR_BAD_CMD);
            END_CASE
        END_IF
    10: // HOME: Z first
        AxZ.HomeExec := TRUE;
        IF AxZ.Sts.homed THEN AxZ.HomeExec := FALSE; iSt := 11; END_IF
    11:
        AxX.HomeExec := TRUE;
        IF AxX.Sts.homed THEN AxX.HomeExec := FALSE; iSt := 12; END_IF
    12:
        AxY.HomeExec := TRUE;
        IF AxY.Sts.homed THEN
            AxY.HomeExec := FALSE; iSt := 0; Busy := FALSE; Done := TRUE;
        END_IF
    20: // position at stroke start, Z up
        AxZ.TargetPos := GVL_Cfg.SC_UP_Z; AxZ.Vel := GVL_Cfg.Z_VEL; AxZ.Acc := GVL_Cfg.Z_ACC;
        AxZ.MoveExec := TRUE;
        IF AxZ.Done THEN AxZ.MoveExec := FALSE; iSt := 21; END_IF
        IF AxZ.Error THEN iSt := 90; END_IF
    21:
        AxX.TargetPos := GVL_Cfg.SC_SWEEP_X0; AxX.Vel := GVL_Cfg.S_VEL; AxX.Acc := GVL_Cfg.S_ACC;
        AxY.TargetPos := GVL_Cfg.SC_ROW_Y[stroke]; AxY.Vel := GVL_Cfg.S_VEL; AxY.Acc := GVL_Cfg.S_ACC;
        AxX.MoveExec := TRUE; AxY.MoveExec := TRUE;
        iSt := 22;
    22:
        IF AxX.Done AND AxY.Done THEN
            AxX.MoveExec := FALSE; AxY.MoveExec := FALSE; iSt := 23;
        END_IF
        IF AxX.Error OR AxY.Error THEN iSt := 90; END_IF
    23: // engage blade
        AxZ.TargetPos := GVL_Cfg.SC_ENGAGE_Z; AxZ.MoveExec := TRUE;
        IF AxZ.Done THEN AxZ.MoveExec := FALSE; iSt := 24; END_IF
        IF AxZ.Error THEN iSt := 90; END_IF
    24: // sweep across
        AxX.TargetPos := GVL_Cfg.SC_SWEEP_X1; AxX.MoveExec := TRUE;
        IF AxX.Done THEN AxX.MoveExec := FALSE; iSt := 25; END_IF
        IF AxX.Error THEN iSt := 90; END_IF
    25: // blade up -> done
        AxZ.TargetPos := GVL_Cfg.SC_UP_Z; AxZ.MoveExec := TRUE;
        IF AxZ.Done THEN
            AxZ.MoveExec := FALSE; iSt := 0; Busy := FALSE; Done := TRUE;
        END_IF
        IF AxZ.Error THEN iSt := 90; END_IF
    60: // PARK
        AxZ.TargetPos := GVL_Cfg.SC_UP_Z; AxZ.MoveExec := TRUE;
        IF AxZ.Done THEN AxZ.MoveExec := FALSE; iSt := 61; END_IF
        IF AxZ.Error THEN iSt := 90; END_IF
    61:
        AxX.TargetPos := 0.0; AxY.TargetPos := 0.0;
        AxX.MoveExec := TRUE; AxY.MoveExec := TRUE;
        IF AxX.Done AND AxY.Done THEN
            AxX.MoveExec := FALSE; AxY.MoveExec := FALSE;
            iSt := 0; Busy := FALSE; Done := TRUE;
        END_IF
        IF AxX.Error OR AxY.Error THEN iSt := 90; END_IF
    90:
        AxX.MoveExec := FALSE; AxY.MoveExec := FALSE; AxZ.MoveExec := FALSE;
        IF ErrorID = 0 THEN
            IF AxX.Error THEN ErrorID := AxX.ErrorID;
            ELSIF AxY.Error THEN ErrorID := AxY.ErrorID;
            ELSIF AxZ.Error THEN ErrorID := AxZ.ErrorID;
            ELSE ErrorID := F_Err(GVL_Cfg.SS_SCRAPER, GVL_Cfg.ERR_DRIVE); END_IF
        END_IF
        iSt := 0; Busy := FALSE; Error := TRUE;
END_CASE
State := TO_UINT(iSt);

END_FUNCTION_BLOCK

// Device/Application/04_L3_Coordination/FB_GriddleTracker
(* ============================================================
   FB_GriddleTracker — per-griddle state + cook timers + HACCP
   record emission. Runs in T_App (called from PRG_JobExec's PRG).
   ScrapeDue fires at cookTime - SCRAPE_GUARD_S so the coordinator
   can stage the scraper. NewHaccp is a LATCHED flag: set here,
   cleared by the consumer (PRG_HACCP, slower task) after reading.
   ============================================================ *)
FUNCTION_BLOCK FB_GriddleTracker
VAR_INPUT
    Sim          : BOOL;
    CycleMs      : LREAL := 20.0;
    // command pulses
    SetLoading   : BOOL;  GIdxA : INT;                 // griddle being loaded
    StartCook    : BOOL;  GIdxB : INT; ItemB : UINT; CountB : INT; BatchB : UDINT;
    ScrapeStart  : BOOL;  GIdxC : INT;
    ScrapeDone   : BOOL;  GIdxD : INT;
    SetFault     : BOOL;  GIdxE : INT;
    HaccpAck     : BOOL;   // consumer (PRG_HACCP) sets after reading the record
END_VAR
VAR_OUTPUT
    aG          : ARRAY[0..3] OF ST_GriddleSts;
    ScrapeDue   : BOOL;
    ScrapeDueG  : INT := -1;
    NewHaccp    : BOOL;
    HaccpRec    : ST_HaccpRec;
END_VAR
VAR
    rtL, rtS, rtP, rtD, rtF : R_TRIG;
    g      : INT;
    dtS    : LREAL;
    rec    : ST_HaccpRec;
    startS : ARRAY[0..3] OF UDINT;
END_VAR

dtS := CycleMs / 1000.0;
IF Sim THEN dtS := dtS * GVL_Cfg.SIM_TIME_SCALE; END_IF
rtL(CLK := SetLoading);  rtS(CLK := StartCook);  rtP(CLK := ScrapeStart);
rtD(CLK := ScrapeDone);  rtF(CLK := SetFault);
// NewHaccp stays latched until the consumer acks it (T_Comms is 5x
// slower than T_App; a 1-cycle pulse would get lost)
IF HaccpAck THEN NewHaccp := FALSE; END_IF

IF rtL.Q AND (GIdxA >= 0) AND (GIdxA <= 3) THEN
    aG[GIdxA].state := TO_UINT(E_GriddleState.LOADING);
END_IF
IF rtS.Q AND (GIdxB >= 0) AND (GIdxB <= 3) THEN
    aG[GIdxB].state := TO_UINT(E_GriddleState.COOKING);
    aG[GIdxB].item  := ItemB;
    aG[GIdxB].count := CountB;
    aG[GIdxB].batchId := BatchB;
    aG[GIdxB].cookElapsedS := 0.0;
    startS[GIdxB] := GVL_Sts.uptimeS;
END_IF
IF rtP.Q AND (GIdxC >= 0) AND (GIdxC <= 3) THEN
    aG[GIdxC].state := TO_UINT(E_GriddleState.SCRAPING);
END_IF
IF rtD.Q AND (GIdxD >= 0) AND (GIdxD <= 3) THEN
    // emit HACCP record, then empty the griddle
    rec.batchId    := aG[GIdxD].batchId;
    rec.item       := aG[GIdxD].item;
    rec.griddleId  := GIdxD;
    rec.platenTopC := GVL_Sts.aHeat[2 * GIdxD].actC;
    rec.platenBotC := GVL_Sts.aHeat[2 * GIdxD + 1].actC;
    rec.cookS      := aG[GIdxD].cookElapsedS;
    rec.tStartS    := startS[GIdxD];
    rec.tEndS      := GVL_Sts.uptimeS;
    IF (rec.platenTopC < GVL_Par.aRecipe[rec.item].platenSetC - 15.0)
       OR (rec.cookS < GVL_Par.aRecipe[rec.item].cookTimeS - 2.0) THEN
        rec.result := 1;    // QUARANTINE
    ELSE
        rec.result := 0;
    END_IF
    HaccpRec := rec; NewHaccp := TRUE;
    aG[GIdxD].state := TO_UINT(E_GriddleState.EMPTY);
    aG[GIdxD].item := 0; aG[GIdxD].count := 0; aG[GIdxD].cookElapsedS := 0.0;
END_IF
IF rtF.Q AND (GIdxE >= 0) AND (GIdxE <= 3) THEN
    aG[GIdxE].state := TO_UINT(E_GriddleState.FAULTED);
END_IF

// cook timers + due flag
ScrapeDue := FALSE; ScrapeDueG := -1;
FOR g := 0 TO 3 DO
    IF aG[g].state = TO_UINT(E_GriddleState.COOKING) THEN
        aG[g].cookElapsedS := aG[g].cookElapsedS + dtS;
        IF aG[g].cookElapsedS >= GVL_Par.aRecipe[aG[g].item].cookTimeS - GVL_Cfg.SCRAPE_GUARD_S THEN
            aG[g].state := TO_UINT(E_GriddleState.READY_TO_SCRAPE);
        END_IF
    END_IF
    IF (aG[g].state = TO_UINT(E_GriddleState.READY_TO_SCRAPE)) AND (ScrapeDueG < 0) THEN
        ScrapeDue := TRUE; ScrapeDueG := g;
    END_IF
    // keep elapsed counting until scraped (for HACCP truth)
    IF aG[g].state = TO_UINT(E_GriddleState.READY_TO_SCRAPE)
       OR aG[g].state = TO_UINT(E_GriddleState.SCRAPING) THEN
        aG[g].cookElapsedS := aG[g].cookElapsedS + dtS;
    END_IF
END_FOR

END_FUNCTION_BLOCK

// Device/Application/04_L3_Coordination/FB_HomingManager
(* ============================================================
   FB_HomingManager — collision-safe machine homing (spec 8.3):
   presses OPEN -> gantry -> scraper -> fork -> griddle carousel
   -> fridge carousel. Runs in T_App (called by PRG_Supervisor,
   which executes BEFORE PRG_Carousels in the task list).
   ============================================================ *)
FUNCTION_BLOCK FB_HomingManager
VAR_INPUT
    Exec  : BOOL;
    Abort : BOOL;
END_VAR
VAR_IN_OUT
    Presses  : ARRAY[0..3] OF FB_Press;
    Gantry   : FB_Gantry;
    Scraper  : FB_Scraper;
    Fork     : FB_Fork;
    GridCar  : FB_GriddleCarousel;
    FridgeCar: FB_FridgeCarousel;
END_VAR
VAR_OUTPUT
    Busy, Done, Error : BOOL;
    ErrorID : UDINT;
    Step    : UINT;
END_VAR
VAR
    iSt : INT;
    i  : INT;
    rtExec : R_TRIG;
    tonTO  : TON;
    allOpen: BOOL;
END_VAR

rtExec(CLK := Exec);
IF Abort THEN iSt := 0; Busy := FALSE; END_IF
tonTO(IN := Busy, PT := T#120S);
IF tonTO.Q AND Busy THEN
    iSt := 0; Busy := FALSE; Error := TRUE;
    ErrorID := F_Err(GVL_Cfg.SS_HOMING, GVL_Cfg.ERR_TIMEOUT);
END_IF

CASE iSt OF
    0:
        IF rtExec.Q THEN
            Done := FALSE; Error := FALSE; ErrorID := 0;
            iSt := 10; Busy := TRUE;
        END_IF
    10: // command all presses HOME (drive re-reference, then open)
        FOR i := 0 TO 3 DO
            Presses[i].Cmd.code := GVL_Cfg.MCMD_HOME;
            Presses[i].CmdExec := TRUE;
        END_FOR
        iSt := 11;
    11:
        allOpen := TRUE;
        FOR i := 0 TO 3 DO
            IF NOT Presses[i].IsOpen THEN allOpen := FALSE; END_IF
            IF Presses[i].Error THEN iSt := 90; ErrorID := Presses[i].ErrorID; END_IF
        END_FOR
        IF allOpen AND (iSt = 11) THEN
            FOR i := 0 TO 3 DO Presses[i].CmdExec := FALSE; END_FOR
            iSt := 20;
        END_IF
    20: // gantry
        Gantry.Cmd.code := GVL_Cfg.MCMD_HOME; Gantry.CmdExec := TRUE;
        iSt := 21;
    21:
        IF Gantry.Done AND Gantry.Homed THEN Gantry.CmdExec := FALSE; iSt := 30; END_IF
        IF Gantry.Error THEN ErrorID := Gantry.ErrorID; iSt := 90; END_IF
    30: // scraper
        Scraper.Cmd.code := GVL_Cfg.MCMD_HOME; Scraper.CmdExec := TRUE;
        iSt := 31;
    31:
        IF Scraper.Done AND Scraper.Homed THEN Scraper.CmdExec := FALSE; iSt := 40; END_IF
        IF Scraper.Error THEN ErrorID := Scraper.ErrorID; iSt := 90; END_IF
    40: // fork
        Fork.Cmd.code := GVL_Cfg.MCMD_HOME; Fork.CmdExec := TRUE;
        iSt := 41;
    41:
        IF Fork.Done AND Fork.Homed THEN Fork.CmdExec := FALSE; iSt := 50; END_IF
        IF Fork.Error THEN ErrorID := Fork.ErrorID; iSt := 90; END_IF
    50: // griddle carousel
        GridCar.HomeExec := TRUE;
        iSt := 51;
    51:
        IF GridCar.Homed THEN GridCar.HomeExec := FALSE; iSt := 60; END_IF
        IF GridCar.Error THEN ErrorID := GridCar.ErrorID; iSt := 90; END_IF
    60: // fridge carousel
        FridgeCar.HomeExec := TRUE;
        iSt := 61;
    61:
        IF FridgeCar.Homed THEN
            FridgeCar.HomeExec := FALSE;
            iSt := 0; Busy := FALSE; Done := TRUE;
        END_IF
        IF FridgeCar.Error THEN ErrorID := FridgeCar.ErrorID; iSt := 90; END_IF
    90:
        Gantry.CmdExec := FALSE; Scraper.CmdExec := FALSE; Fork.CmdExec := FALSE;
        GridCar.HomeExec := FALSE; FridgeCar.HomeExec := FALSE;
        FOR i := 0 TO 3 DO Presses[i].CmdExec := FALSE; END_FOR
        iSt := 0; Busy := FALSE; Error := TRUE;
END_CASE
Step := TO_UINT(iSt);

END_FUNCTION_BLOCK

// Device/Application/04_L3_Coordination/FB_JobQueue
(* ============================================================
   FB_JobQueue — ring buffer of ST_PattyJob (size 64).
   ============================================================ *)
FUNCTION_BLOCK FB_JobQueue
VAR_INPUT
    PushExec : BOOL;
    JobIn    : ST_PattyJob;
    PopExec  : BOOL;
    ClearExec: BOOL;
END_VAR
VAR_OUTPUT
    JobOut : ST_PattyJob;
    Count  : INT;
    Full   : BOOL;
    Empty  : BOOL;
    PopOk  : BOOL;
END_VAR
VAR
    buf  : ARRAY[0..63] OF ST_PattyJob;
    head : INT;   // next write
    tail : INT;   // next read
    rtPush, rtPop, rtClr : R_TRIG;
END_VAR

rtPush(CLK := PushExec);
rtPop(CLK := PopExec);
rtClr(CLK := ClearExec);
IF rtClr.Q THEN head := 0; tail := 0; Count := 0; END_IF
Full  := Count >= 64;
Empty := Count = 0;
PopOk := FALSE;
IF rtPush.Q AND NOT Full THEN
    buf[head] := JobIn;
    head := (head + 1) MOD 64;
    Count := Count + 1;
END_IF
IF rtPop.Q AND NOT Empty THEN
    JobOut := buf[tail];
    tail := (tail + 1) MOD 64;
    Count := Count - 1;
    PopOk := TRUE;
END_IF

END_FUNCTION_BLOCK
